C03646=1227.699,20.844,-42.507,-179.267,5.370,148.713
C03647=1227.694,21.094,-42.523,-179.265,5.371,148.713
C03648=1227.689,21.344,-42.538,-179.262,5.371,148.712
C03649=1227.684,21.593,-42.554,-179.259,5.372,148.711
C03650=1227.679,21.842,-42.569,-179.257,5.372,148.711
C03651=1227.674,22.092,-42.584,-179.255,5.372,148.710
C03652=1227.669,22.342,-42.600,-179.252,5.373,148.709
C03653=1227.664,22.591,-42.615,-179.250,5.373,148.709
C03654=1227.659,22.841,-42.630,-179.247,5.374,148.708
C03655=1227.654,23.090,-42.645,-179.244,5.374,148.707
C03656=1227.649,23.339,-42.661,-179.242,5.375,148.707
C03657=1227.644,23.589,-42.677,-179.240,5.375,148.706
C03658=1227.639,23.838,-42.692,-179.237,5.375,148.705
C03659=1227.634,24.088,-42.707,-179.234,5.376,148.705
C03660=1227.629,24.337,-42.722,-179.232,5.376,148.704
C03661=1227.625,24.587,-42.738,-179.229,5.377,148.703
C03662=1227.619,24.836,-42.754,-179.227,5.377,148.703
C03663=1227.615,25.085,-42.769,-179.224,5.377,148.702
C03664=1227.609,25.335,-42.784,-179.222,5.378,148.701
C03665=1227.604,25.585,-42.800,-179.219,5.378,148.701
C03666=1227.600,25.834,-42.815,-179.216,5.379,148.700
C03667=1227.594,26.083,-42.831,-179.214,5.379,148.699
C03668=1227.589,26.333,-42.847,-179.212,5.379,148.699
C03669=1227.585,26.583,-42.862,-179.209,5.380,148.698
C03670=1227.579,26.832,-42.878,-179.206,5.380,148.697
C03671=1227.574,27.081,-42.893,-179.204,5.381,148.697
C03672=1227.569,27.330,-42.908,-179.202,5.382,148.696
C03673=1227.565,27.581,-42.924,-179.199,5.382,148.695
C03674=1227.559,27.830,-42.940,-179.197,5.382,148.695
C03675=1227.554,28.079,-42.955,-179.194,5.382,148.694
C03676=1227.550,28.329,-42.971,-179.192,5.383,148.693
C03677=1227.544,28.579,-42.986,-179.189,5.384,148.693
C03678=1227.539,28.827,-43.002,-179.186,5.384,148.692
C03679=1227.535,29.076,-43.017,-179.184,5.385,148.691
C03680=1227.530,29.346,-43.035,-179.181,5.385,148.691
C03681=1227.524,29.615,-43.051,-179.178,5.386,148.690
C03682=1227.518,29.883,-43.068,-179.176,5.386,148.689
C03683=1227.513,30.152,-43.085,-179.173,5.387,148.688
C03684=1227.508,30.401,-43.100,-179.171,5.386,148.688
C03685=1227.503,30.651,-43.116,-179.168,5.387,148.687
C03686=1227.498,30.900,-43.132,-179.166,5.388,148.687
C03687=1227.493,31.149,-43.148,-179.163,5.388,148.686
C03688=1227.488,31.399,-43.164,-179.161,5.389,148.685
C03689=1227.483,31.648,-43.179,-179.158,5.389,148.684
C03690=1227.478,31.898,-43.195,-179.155,5.390,148.684
C03691=1227.474,32.147,-43.211,-179.153,5.390,148.683
C03692=1227.468,32.397,-43.227,-179.151,5.390,148.682
C03693=1227.463,32.647,-43.243,-179.148,5.391,148.682
C03694=1227.459,32.896,-43.258,-179.145,5.391,148.681
C03695=1227.454,33.145,-43.274,-179.143,5.392,148.680
C03696=1227.449,33.395,-43.290,-179.140,5.392,148.680
C03697=1227.444,33.644,-43.306,-179.137,5.393,148.679
C03698=1227.438,33.893,-43.321,-179.135,5.393,148.678
C03699=1227.434,34.143,-43.338,-179.133,5.393,148.678
C03700=1227.429,34.392,-43.353,-179.130,5.394,148.677
C03701=1227.424,34.642,-43.369,-179.128,5.395,148.677
C03702=1227.419,34.891,-43.385,-179.125,5.395,148.676
C03703=1227.414,35.140,-43.401,-179.123,5.396,148.675
C03704=1227.409,35.390,-43.417,-179.120,5.396,148.675
C03705=1227.404,35.640,-43.432,-179.118,5.396,148.674
C03706=1227.399,35.889,-43.449,-179.115,5.397,148.673
C03707=1227.394,36.139,-43.465,-179.113,5.397,148.673
C03708=1227.389,36.387,-43.480,-179.110,5.398,148.672
C03709=1227.385,36.637,-43.496,-179.107,5.398,148.671
C03710=1227.379,36.887,-43.512,-179.105,5.399,148.671
C03711=1227.375,37.136,-43.528,-179.102,5.399,148.670
C03712=1227.369,37.386,-43.544,-179.100,5.400,148.669
C03713=1227.364,37.635,-43.560,-179.098,5.400,148.669
C03714=1227.359,37.884,-43.576,-179.095,5.401,148.668
C03715=1227.354,38.134,-43.592,-179.092,5.401,148.667
C03716=1227.350,38.383,-43.609,-179.090,5.402,148.667
C03717=1227.344,38.633,-43.624,-179.087,5.402,148.666
C03718=1227.339,38.883,-43.640,-179.085,5.403,148.665
C03719=1227.334,39.132,-43.656,-179.082,5.403,148.665
C03720=1227.330,39.382,-43.672,-179.079,5.404,148.664
C03721=1227.324,39.631,-43.689,-179.077,5.405,148.663
C03722=1227.319,39.880,-43.704,-179.075,5.404,148.663
C03723=1227.315,40.129,-43.721,-179.072,5.405,148.662
C03724=1227.309,40.379,-43.736,-179.070,5.406,148.662
C03725=1227.305,40.628,-43.753,-179.067,5.406,148.661
C03726=1227.299,40.878,-43.769,-179.064,5.407,148.660
C03727=1227.295,41.127,-43.785,-179.062,5.407,148.659
C03728=1227.289,41.377,-43.801,-179.059,5.408,148.659
C03729=1227.285,41.626,-43.818,-179.057,5.409,148.658
C03730=1227.280,41.875,-43.833,-179.054,5.409,148.657
C03731=1227.275,42.125,-43.850,-179.052,5.409,148.657
C03732=1227.270,42.374,-43.866,-179.049,5.409,148.656
C03733=1227.265,42.624,-43.882,-179.047,5.410,148.655
C03734=1227.260,42.873,-43.898,-179.044,5.411,148.655
C03735=1227.255,43.123,-43.914,-179.042,5.411,148.654
C03736=1227.250,43.372,-43.931,-179.039,5.412,148.654
C03737=1227.246,43.622,-43.947,-179.037,5.413,148.653
C03738=1227.240,43.870,-43.963,-179.034,5.413,148.652
C03739=1227.236,44.120,-43.980,-179.031,5.414,148.652
C03740=1227.230,44.370,-43.996,-179.029,5.414,148.651
C03741=1227.225,44.619,-44.013,-179.027,5.414,148.650
C03742=1227.221,44.869,-44.028,-179.024,5.415,148.650
C03743=1227.215,45.118,-44.045,-179.022,5.416,148.649
C03744=1227.211,45.367,-44.061,-179.019,5.416,148.649
C03745=1227.206,45.617,-44.077,-179.016,5.417,148.648
C03746=1227.201,45.866,-44.094,-179.014,5.417,148.647
C03747=1227.196,46.115,-44.110,-179.011,5.418,148.646
C03748=1227.191,46.365,-44.126,-179.009,5.418,148.646
C03749=1227.185,46.614,-44.143,-179.006,5.419,148.645
C03750=1227.181,46.864,-44.160,-179.003,5.419,148.644
C03751=1227.176,47.114,-44.175,-179.001,5.420,148.644
C03752=1227.171,47.363,-44.192,-178.998,5.421,148.643
C03753=1227.167,47.612,-44.208,-178.996,5.421,148.643
C03754=1227.162,47.861,-44.225,-178.994,5.421,148.642
C03755=1227.157,48.111,-44.241,-178.991,5.422,148.641
C03756=1227.151,48.360,-44.258,-178.989,5.422,148.641
C03757=1227.146,48.610,-44.274,-178.986,5.423,148.640
C03758=1227.142,48.859,-44.291,-178.983,5.424,148.639
C03759=1227.137,49.109,-44.307,-178.981,5.424,148.639
C03760=1227.132,49.358,-44.323,-178.978,5.425,148.638
C03761=1227.127,49.608,-44.340,-178.976,5.426,148.638
C03762=1227.122,49.857,-44.357,-178.973,5.426,148.637
C03763=1227.117,50.106,-44.373,-178.971,5.427,148.636
C03764=1227.112,50.355,-44.389,-178.968,5.427,148.636
C03765=1227.107,50.605,-44.406,-178.965,5.428,148.635
C03766=1227.102,50.855,-44.423,-178.963,5.428,148.634
C03767=1227.097,51.104,-44.439,-178.961,5.428,148.634
C03768=1227.093,51.353,-44.456,-178.958,5.429,148.633
C03769=1227.088,51.603,-44.473,-178.956,5.430,148.632
C03770=1227.082,51.852,-44.490,-178.953,5.430,148.632
C03771=1227.078,52.102,-44.505,-178.951,5.431,148.631
C03772=1227.073,52.351,-44.522,-178.948,5.431,148.630
C03773=1227.067,52.600,-44.539,-178.945,5.432,148.630
C03774=1227.063,52.850,-44.556,-178.943,5.433,148.629
C03775=1227.058,53.099,-44.572,-178.940,5.433,148.628
C03776=1227.053,53.348,-44.589,-178.938,5.434,148.628
C03777=1227.048,53.598,-44.606,-178.935,5.435,148.627
C03778=1227.044,53.847,-44.623,-178.933,5.435,148.627
C03779=1227.038,54.096,-44.639,-178.930,5.436,148.626
C03780=1227.033,54.346,-44.656,-178.927,5.436,148.625
C03781=1227.029,54.595,-44.673,-178.925,5.437,148.625
C03782=1227.024,54.844,-44.689,-178.922,5.437,148.624
C03783=1227.019,55.094,-44.706,-178.920,5.438,148.624
C03784=1227.013,55.362,-44.723,-178.917,5.439,148.623
C03785=1227.008,55.631,-44.742,-178.914,5.439,148.622
C03786=1227.002,55.899,-44.760,-178.911,5.440,148.621
C03787=1226.998,56.168,-44.778,-178.909,5.440,148.621
C03788=1226.992,56.418,-44.795,-178.906,5.441,148.620
C03789=1226.987,56.666,-44.812,-178.904,5.441,148.619
C03790=1226.983,56.916,-44.828,-178.901,5.442,148.619
C03791=1226.978,57.166,-44.845,-178.899,5.443,148.618
C03792=1226.973,57.415,-44.862,-178.896,5.444,148.618
C03793=1226.967,57.664,-44.879,-178.894,5.444,148.617
C03794=1226.963,57.914,-44.896,-178.891,5.445,148.616
C03795=1226.958,58.163,-44.912,-178.888,5.445,148.616
C03796=1226.953,58.413,-44.930,-178.886,5.446,148.615
C03797=1226.948,58.662,-44.946,-178.883,5.447,148.614
C03798=1226.943,58.911,-44.964,-178.881,5.447,148.614
C03799=1226.939,59.160,-44.981,-178.878,5.448,148.613
C03800=1226.933,59.410,-44.998,-178.876,5.448,148.612
C03801=1226.928,59.659,-45.014,-178.873,5.449,148.612
C03802=1226.924,59.908,-45.031,-178.870,5.450,148.611
C03803=1226.919,60.158,-45.048,-178.868,5.451,148.611
C03804=1226.914,60.408,-45.065,-178.866,5.451,148.610
C03805=1226.909,60.656,-45.082,-178.863,5.452,148.609
C03806=1226.904,60.906,-45.099,-178.860,5.452,148.609
C03807=1226.899,61.155,-45.116,-178.858,5.453,148.608
C03808=1226.895,61.405,-45.133,-178.855,5.453,148.607
C03809=1226.889,61.655,-45.150,-178.853,5.454,148.607
C03810=1226.884,61.904,-45.167,-178.851,5.454,148.606
C03811=1226.879,62.153,-45.185,-178.848,5.455,148.606
C03812=1226.875,62.402,-45.201,-178.846,5.455,148.605
C03813=1226.870,62.652,-45.218,-178.843,5.456,148.604
C03814=1226.865,62.901,-45.235,-178.840,5.456,148.604
C03815=1226.860,63.150,-45.253,-178.838,5.457,148.603
C03816=1226.855,63.399,-45.269,-178.836,5.458,148.602
C03817=1226.850,63.649,-45.287,-178.833,5.459,148.602
C03818=1226.845,63.899,-45.303,-178.830,5.459,148.601
C03819=1226.841,64.148,-45.321,-178.828,5.460,148.600
C03820=1226.835,64.398,-45.339,-178.825,5.461,148.600
C03821=1226.830,64.646,-45.355,-178.823,5.461,148.599
C03822=1226.825,64.896,-45.373,-178.820,5.462,148.599
C03823=1226.821,65.145,-45.390,-178.818,5.462,148.598
C03824=1226.816,65.395,-45.407,-178.815,5.463,148.597
C03825=1226.811,65.644,-45.424,-178.812,5.463,148.597
C03826=1226.806,65.894,-45.441,-178.810,5.464,148.596
C03827=1226.801,66.143,-45.459,-178.808,5.465,148.596
C03828=1226.796,66.392,-45.476,-178.805,5.466,148.595
C03829=1226.791,66.641,-45.493,-178.802,5.466,148.594
C03830=1226.787,66.891,-45.510,-178.800,5.467,148.594
C03831=1226.782,67.140,-45.528,-178.798,5.468,148.593
C03832=1226.776,67.390,-45.545,-178.794,5.469,148.593
C03833=1226.772,67.639,-45.562,-178.792,5.470,148.592
C03834=1226.767,67.888,-45.580,-178.789,5.470,148.591
C03835=1226.762,68.138,-45.597,-178.786,5.471,148.591
C03836=1226.757,68.386,-45.614,-178.784,5.471,148.590
C03837=1226.752,68.636,-45.631,-178.782,5.472,148.589
C03838=1226.747,68.885,-45.649,-178.779,5.473,148.589
C03839=1226.742,69.135,-45.666,-178.776,5.474,148.588
C03840=1226.738,69.384,-45.684,-178.774,5.474,148.587
C03841=1226.732,69.634,-45.701,-178.771,5.475,148.587
C03842=1226.728,69.883,-45.718,-178.769,5.476,148.586
C03843=1226.723,70.132,-45.736,-178.766,5.476,148.586
C03844=1226.718,70.382,-45.753,-178.764,5.477,148.585
C03845=1226.714,70.631,-45.770,-178.761,5.477,148.584
C03846=1226.709,70.880,-45.788,-178.758,5.478,148.584
C03847=1226.703,71.130,-45.806,-178.756,5.479,148.583
C03848=1226.699,71.379,-45.823,-178.754,5.479,148.583
C03849=1226.694,71.629,-45.840,-178.751,5.480,148.582
C03850=1226.688,71.877,-45.858,-178.748,5.481,148.581
C03851=1226.683,72.127,-45.875,-178.746,5.481,148.581
C03852=1226.679,72.376,-45.892,-178.744,5.482,148.580
C03853=1226.674,72.626,-45.910,-178.741,5.483,148.580
C03854=1226.669,72.875,-45.928,-178.738,5.483,148.579
C03855=1226.664,73.125,-45.945,-178.736,5.484,148.578
C03856=1226.660,73.374,-45.962,-178.733,5.485,148.578
C03857=1226.655,73.623,-45.980,-178.731,5.485,148.577
C03858=1226.649,73.873,-45.998,-178.728,5.486,148.577
C03859=1226.645,74.122,-46.016,-178.726,5.487,148.576
C03860=1226.640,74.371,-46.034,-178.723,5.487,148.575
C03861=1226.635,74.620,-46.050,-178.721,5.488,148.575
C03862=1226.630,74.870,-46.068,-178.718,5.490,148.574
C03863=1226.625,75.119,-46.086,-178.715,5.490,148.573
C03864=1226.620,75.368,-46.103,-178.713,5.491,148.573
C03865=1226.615,75.618,-46.121,-178.710,5.491,148.572
C03866=1226.610,75.867,-46.139,-178.708,5.492,148.572
C03867=1226.606,76.116,-46.156,-178.705,5.493,148.571
C03868=1226.601,76.366,-46.174,-178.703,5.493,148.570
C03869=1226.596,76.615,-46.192,-178.700,5.494,148.570
C03870=1226.591,76.864,-46.209,-178.698,5.495,148.569
C03871=1226.586,77.114,-46.227,-178.695,5.496,148.569
C03872=1226.581,77.363,-46.245,-178.693,5.496,148.568
C03873=1226.577,77.612,-46.263,-178.690,5.497,148.567
C03874=1226.572,77.861,-46.280,-178.687,5.497,148.567
C03875=1226.567,78.111,-46.298,-178.685,5.498,148.566
C03876=1226.562,78.361,-46.316,-178.683,5.499,148.566
C03877=1226.557,78.610,-46.334,-178.680,5.499,148.565
C03878=1226.552,78.860,-46.351,-178.677,5.500,148.564
C03879=1226.547,79.109,-46.369,-178.675,5.502,148.564
C03880=1226.542,79.358,-46.387,-178.672,5.502,148.563
C03881=1226.537,79.607,-46.405,-178.669,5.503,148.563
C03882=1226.533,79.856,-46.423,-178.667,5.504,148.562
C03883=1226.527,80.106,-46.441,-178.665,5.505,148.561
C03884=1226.522,80.355,-46.459,-178.662,5.505,148.561
C03885=1226.518,80.604,-46.476,-178.659,5.506,148.560
C03886=1226.513,80.853,-46.494,-178.657,5.506,148.559
C03887=1226.508,81.102,-46.512,-178.655,5.507,148.559
C03888=1226.503,81.371,-46.531,-178.652,5.508,148.558
C03889=1226.497,81.640,-46.551,-178.649,5.509,148.558
C03890=1226.492,81.908,-46.570,-178.646,5.510,148.557
C03891=1226.487,82.176,-46.589,-178.643,5.510,148.556
C03892=1226.482,82.426,-46.607,-178.641,5.511,148.556
C03893=1226.477,82.675,-46.625,-178.638,5.512,148.555
C03894=1226.473,82.925,-46.644,-178.636,5.512,148.554
C03895=1226.468,83.174,-46.662,-178.633,5.514,148.554
C03896=1226.463,83.423,-46.680,-178.630,5.515,148.553
C03897=1226.458,83.672,-46.698,-178.628,5.515,148.553
C03898=1226.453,83.921,-46.716,-178.625,5.516,148.552
C03899=1226.448,84.170,-46.734,-178.623,5.517,148.552
C03900=1226.443,84.420,-46.752,-178.620,5.517,148.551
C03901=1226.439,84.670,-46.770,-178.618,5.518,148.550
C03902=1226.434,84.919,-46.788,-178.616,5.519,148.550
C03903=1226.429,85.168,-46.806,-178.613,5.519,148.549
C03904=1226.424,85.417,-46.824,-178.610,5.520,148.549
C03905=1226.419,85.666,-46.842,-178.607,5.522,148.548
C03906=1226.415,85.915,-46.860,-178.605,5.522,148.548
C03907=1226.410,86.165,-46.878,-178.602,5.523,148.547
C03908=1226.405,86.414,-46.896,-178.600,5.524,148.546
C03909=1226.400,86.664,-46.914,-178.597,5.524,148.546
C03910=1226.395,86.913,-46.933,-178.595,5.525,148.545
C03911=1226.390,87.162,-46.951,-178.592,5.526,148.545
C03912=1226.385,87.411,-46.969,-178.590,5.526,148.544
C03913=1226.381,87.661,-46.987,-178.587,5.527,148.543
C03914=1226.376,87.911,-47.005,-178.584,5.529,148.543
C03915=1226.371,88.160,-47.023,-178.582,5.529,148.542
C03916=1226.366,88.408,-47.042,-178.579,5.530,148.541
C03917=1226.361,88.657,-47.060,-178.577,5.531,148.541
C03918=1226.356,88.908,-47.079,-178.574,5.532,148.540
C03919=1226.351,89.157,-47.097,-178.572,5.532,148.540
C03920=1226.346,89.406,-47.115,-178.569,5.533,148.539
C03921=1226.342,89.655,-47.133,-178.567,5.534,148.539
C03922=1226.337,89.905,-47.151,-178.564,5.535,148.538
C03923=1226.333,90.154,-47.170,-178.561,5.536,148.537
C03924=1226.327,90.403,-47.188,-178.559,5.537,148.537
C03925=1226.322,90.652,-47.206,-178.556,5.537,148.536
C03926=1226.318,90.902,-47.225,-178.554,5.538,148.536
C03927=1226.313,91.151,-47.243,-178.551,5.538,148.535
C03928=1226.308,91.400,-47.261,-178.549,5.539,148.535
C03929=1226.303,91.649,-47.280,-178.546,5.540,148.534
C03930=1226.298,91.899,-47.298,-178.543,5.541,148.533
C03931=1226.293,92.148,-47.316,-178.541,5.542,148.533
C03932=1226.289,92.397,-47.335,-178.539,5.543,148.532
C03933=1226.283,92.646,-47.353,-178.536,5.544,148.532
C03934=1226.279,92.896,-47.372,-178.533,5.544,148.531
C03935=1226.274,93.145,-47.390,-178.531,5.545,148.531
C03936=1226.269,93.394,-47.408,-178.529,5.546,148.530
C03937=1226.264,93.644,-47.427,-178.525,5.547,148.529
C03938=1226.259,93.893,-47.445,-178.523,5.548,148.529
C03939=1226.255,94.142,-47.464,-178.521,5.549,148.528
C03940=1226.250,94.391,-47.482,-178.518,5.549,148.527
C03941=1226.245,94.641,-47.501,-178.516,5.550,148.527
C03942=1226.240,94.890,-47.520,-178.513,5.551,148.526
C03943=1226.235,95.139,-47.538,-178.510,5.552,148.526
C03944=1226.230,95.389,-47.557,-178.507,5.553,148.525
C03945=1226.226,95.638,-47.575,-178.505,5.554,148.525
C03946=1226.221,95.887,-47.593,-178.503,5.554,148.524
C03947=1226.217,96.136,-47.612,-178.500,5.555,148.523
C03948=1226.211,96.386,-47.631,-178.498,5.556,148.523
C03949=1226.206,96.634,-47.650,-178.495,5.557,148.522
C03950=1226.201,96.884,-47.669,-178.492,5.558,148.522
C03951=1226.196,97.134,-47.687,-178.490,5.559,148.521
C03952=1226.192,97.382,-47.705,-178.487,5.560,148.521
C03953=1226.187,97.632,-47.724,-178.485,5.560,148.520
C03954=1226.182,97.881,-47.743,-178.483,5.561,148.520
C03955=1226.177,98.130,-47.761,-178.480,5.562,148.519
C03956=1226.172,98.380,-47.780,-178.477,5.563,148.518
C03957=1226.168,98.629,-47.798,-178.475,5.564,148.518
C03958=1226.163,98.878,-47.818,-178.472,5.565,148.517
C03959=1226.158,99.128,-47.836,-178.470,5.565,148.517
C03960=1226.153,99.376,-47.855,-178.467,5.566,148.516
C03961=1226.148,99.626,-47.874,-178.464,5.568,148.516
C03962=1226.144,99.875,-47.892,-178.462,5.568,148.515
C03963=1226.139,100.125,-47.911,-178.459,5.569,148.514
C03964=1226.134,100.374,-47.930,-178.457,5.570,148.514
C03965=1226.129,100.623,-47.948,-178.454,5.571,148.513
C03966=1226.124,100.872,-47.968,-178.452,5.572,148.513
C03967=1226.120,101.121,-47.986,-178.449,5.573,148.512
C03968=1226.115,101.371,-48.005,-178.446,5.574,148.511
C03969=1226.110,101.620,-48.024,-178.444,5.575,148.511
C03970=1226.104,101.869,-48.043,-178.442,5.575,148.510
C03971=1226.100,102.118,-48.062,-178.439,5.576,148.510
C03972=1226.095,102.367,-48.081,-178.436,5.578,148.509
C03973=1226.091,102.617,-48.099,-178.434,5.578,148.509
C03974=1226.085,102.866,-48.119,-178.431,5.579,148.508
C03975=1226.081,103.115,-48.138,-178.429,5.580,148.508
C03976=1226.076,103.365,-48.156,-178.426,5.580,148.507
C03977=1226.071,103.613,-48.175,-178.423,5.582,148.506
C03978=1226.066,103.863,-48.195,-178.421,5.583,148.506
C03979=1226.062,104.112,-48.213,-178.418,5.583,148.505
C03980=1226.057,104.362,-48.232,-178.416,5.584,148.505
C03981=1226.052,104.610,-48.251,-178.414,5.585,148.504
C03982=1226.047,104.860,-48.270,-178.410,5.586,148.504
C03983=1226.043,105.109,-48.289,-178.408,5.587,148.503
C03984=1226.038,105.359,-48.308,-178.406,5.588,148.503
C03985=1226.033,105.607,-48.327,-178.403,5.589,148.502
C03986=1226.028,105.857,-48.346,-178.401,5.589,148.501
C03987=1226.023,106.106,-48.365,-178.398,5.591,148.501
C03988=1226.019,106.355,-48.384,-178.395,5.592,148.500
C03989=1226.013,106.604,-48.403,-178.393,5.592,148.500
C03990=1226.009,106.854,-48.422,-178.390,5.593,148.499
C03991=1226.004,107.103,-48.441,-178.387,5.595,148.499
C03992=1225.999,107.372,-48.462,-178.385,5.595,148.498
C03993=1225.993,107.640,-48.483,-178.383,5.596,148.497
C03994=1225.989,107.909,-48.503,-178.379,5.598,148.497
C03995=1225.983,108.176,-48.523,-178.377,5.598,148.496
C03996=1225.979,108.426,-48.543,-178.374,5.599,148.496
C03997=1225.973,108.675,-48.562,-178.371,5.601,148.495
C03998=1225.969,108.925,-48.581,-178.369,5.601,148.495
C03999=1225.964,109.174,-48.600,-178.367,5.602,148.494
C04000=1225.959,109.423,-48.620,-178.364,5.603,148.493
C04001=1225.954,109.672,-48.638,-178.361,5.604,148.493
C04002=1225.950,109.921,-48.658,-178.359,5.605,148.492
C04003=1225.945,110.171,-48.678,-178.356,5.606,148.492
C04004=1225.940,110.419,-48.696,-178.354,5.606,148.491
C04005=1225.935,110.669,-48.716,-178.351,5.607,148.491
C04006=1225.930,110.918,-48.735,-178.348,5.609,148.490
C04007=1225.926,111.167,-48.754,-178.346,5.610,148.490
C04008=1225.921,111.416,-48.774,-178.344,5.610,148.489
C04009=1225.916,111.666,-48.793,-178.341,5.611,148.488
C04010=1225.912,111.915,-48.812,-178.338,5.613,148.488
C04011=1225.907,112.164,-48.832,-178.336,5.613,148.487
C04012=1225.902,112.413,-48.851,-178.333,5.614,148.487
C04013=1225.897,112.662,-48.871,-178.331,5.615,148.486
C04014=1225.893,112.911,-48.890,-178.328,5.616,148.486
C04015=1225.888,113.161,-48.909,-178.326,5.617,148.485
C04016=1225.882,113.410,-48.929,-178.323,5.618,148.485
C04017=1225.878,113.659,-48.948,-178.321,5.619,148.484
C04018=1225.873,113.908,-48.967,-178.318,5.620,148.484
C04019=1225.868,114.158,-48.987,-178.315,5.621,148.483
C04020=1225.864,114.407,-49.006,-178.313,5.622,148.483
C04021=1225.858,114.656,-49.026,-178.310,5.623,148.482
C04022=1225.854,114.906,-49.045,-178.308,5.624,148.481
C04023=1225.849,115.154,-49.064,-178.305,5.625,148.481
C04024=1225.844,115.404,-49.084,-178.302,5.626,148.480
C04025=1225.839,115.653,-49.103,-178.300,5.627,148.480
C04026=1225.834,115.902,-49.123,-178.297,5.628,148.479
C04027=1225.829,116.152,-49.142,-178.295,5.629,148.479
C04028=1225.825,116.401,-49.163,-178.292,5.630,148.478
C04029=1225.820,116.649,-49.181,-178.289,5.631,148.477
C04030=1225.816,116.899,-49.201,-178.287,5.632,148.477
C04031=1225.811,117.148,-49.221,-178.284,5.633,148.476
C04032=1225.805,117.397,-49.240,-178.282,5.634,148.476
C04033=1225.801,117.647,-49.260,-178.279,5.635,148.475
C04034=1225.796,117.896,-49.280,-178.277,5.636,148.475
C04035=1225.791,118.145,-49.299,-178.274,5.637,148.474
C04036=1225.786,118.394,-49.319,-178.271,5.638,148.474
C04037=1225.782,118.643,-49.338,-178.269,5.639,148.473
C04038=1225.777,118.892,-49.357,-178.267,5.640,148.473
C04039=1225.772,119.141,-49.378,-178.264,5.641,148.472
C04040=1225.768,119.391,-49.397,-178.261,5.642,148.472
C04041=1225.763,119.640,-49.417,-178.259,5.643,148.471
C04042=1225.758,119.889,-49.436,-178.257,5.644,148.471
C04043=1225.753,120.138,-49.457,-178.253,5.645,148.470
C04044=1225.748,120.388,-49.476,-178.251,5.646,148.470
C04045=1225.743,120.637,-49.495,-178.249,5.647,148.469
C04046=1225.739,120.886,-49.516,-178.246,5.649,148.469
C04047=1225.734,121.135,-49.536,-178.243,5.649,148.468
C04048=1225.729,121.385,-49.555,-178.241,5.650,148.467
C04049=1225.724,121.633,-49.575,-178.239,5.651,148.467
C04050=1225.719,121.883,-49.595,-178.235,5.652,148.466
C04051=1225.715,122.132,-49.614,-178.233,5.653,148.466
C04052=1225.710,122.381,-49.635,-178.231,5.654,148.465
C04053=1225.705,122.630,-49.654,-178.228,5.656,148.465
C04054=1225.700,122.879,-49.674,-178.225,5.656,148.464
C04055=1225.696,123.128,-49.694,-178.223,5.657,148.464
C04056=1225.691,123.378,-49.714,-178.220,5.659,148.463
C04057=1225.686,123.626,-49.734,-178.218,5.660,148.463
C04058=1225.681,123.876,-49.753,-178.215,5.660,148.462
C04059=1225.676,124.125,-49.773,-178.212,5.662,148.461
C04060=1225.672,124.374,-49.794,-178.210,5.663,148.461
C04061=1225.667,124.624,-49.813,-178.208,5.663,148.460
C04062=1225.662,124.872,-49.833,-178.205,5.664,148.460
C04063=1225.657,125.122,-49.853,-178.202,5.666,148.459
C04064=1225.653,125.371,-49.873,-178.200,5.667,148.459
C04065=1225.648,125.620,-49.893,-178.198,5.667,148.458
C04066=1225.644,125.869,-49.913,-178.195,5.669,148.458
C04067=1225.638,126.118,-49.933,-178.192,5.670,148.457
C04068=1225.634,126.367,-49.953,-178.190,5.671,148.457
C04069=1225.629,126.617,-49.973,-178.187,5.672,148.456
C04070=1225.625,126.865,-49.993,-178.185,5.673,148.456
C04071=1225.620,127.115,-50.013,-178.182,5.674,148.455
C04072=1225.615,127.364,-50.034,-178.179,5.675,148.455
C04073=1225.610,127.613,-50.053,-178.177,5.676,148.454
C04074=1225.605,127.862,-50.073,-178.174,5.677,148.454
C04075=1225.600,128.112,-50.093,-178.172,5.679,148.453
C04076=1225.596,128.361,-50.113,-178.169,5.679,148.453
C04077=1225.592,128.610,-50.134,-178.167,5.680,148.452
C04078=1225.587,128.859,-50.153,-178.164,5.682,148.452
C04079=1225.581,129.108,-50.174,-178.162,5.683,148.451
C04080=1225.576,129.357,-50.194,-178.159,5.684,148.451
C04081=1225.572,129.606,-50.214,-178.156,5.685,148.450
C04082=1225.567,129.855,-50.234,-178.154,5.686,148.449
C04083=1225.563,130.105,-50.254,-178.151,5.688,148.449
C04084=1225.558,130.354,-50.274,-178.149,5.688,148.448
C04085=1225.553,130.603,-50.295,-178.146,5.689,148.448
C04086=1225.548,130.853,-50.315,-178.143,5.691,148.447
C04087=1225.544,131.101,-50.335,-178.141,5.692,148.447
C04088=1225.539,131.350,-50.355,-178.139,5.692,148.446
C04089=1225.534,131.599,-50.375,-178.136,5.694,148.446
C04090=1225.529,131.849,-50.396,-178.133,5.695,148.445
C04091=1225.524,132.098,-50.416,-178.131,5.696,148.445
C04092=1225.520,132.346,-50.437,-178.128,5.697,148.444
C04093=1225.515,132.596,-50.456,-178.126,5.698,148.444
C04094=1225.510,132.845,-50.477,-178.123,5.700,148.443
C04095=1225.506,133.094,-50.498,-178.121,5.701,148.443
C04096=1225.500,133.363,-50.519,-178.118,5.701,148.442
C04097=1225.495,133.631,-50.541,-178.115,5.703,148.442
C04098=1225.490,133.900,-50.563,-178.112,5.705,148.441
C04099=1225.485,134.169,-50.586,-178.110,5.705,148.441
C04100=1225.481,134.418,-50.606,-178.106,5.707,148.440
C04101=1225.476,134.667,-50.626,-178.104,5.708,148.440
C04102=1225.471,134.916,-50.647,-178.102,5.708,148.439
C04103=1225.466,135.165,-50.667,-178.099,5.710,148.439
C04104=1225.461,135.414,-50.687,-178.096,5.711,148.438
C04105=1225.456,135.663,-50.708,-178.094,5.712,148.438
C04106=1225.452,135.912,-50.728,-178.092,5.713,148.437
C04107=1225.447,136.161,-50.749,-178.089,5.714,148.437
C04108=1225.442,136.411,-50.770,-178.086,5.716,148.436
C04109=1225.438,136.660,-50.790,-178.084,5.717,148.436
C04110=1225.433,136.909,-50.810,-178.082,5.717,148.435
C04111=1225.428,137.158,-50.831,-178.078,5.719,148.435
C04112=1225.423,137.407,-50.851,-178.076,5.720,148.434
C04113=1225.419,137.656,-50.871,-178.073,5.721,148.434
C04114=1225.414,137.906,-50.892,-178.071,5.722,148.433
C04115=1225.409,138.155,-50.913,-178.068,5.723,148.433
C04116=1225.404,138.404,-50.934,-178.066,5.725,148.432
C04117=1225.400,138.653,-50.954,-178.063,5.725,148.432
C04118=1225.394,138.902,-50.975,-178.061,5.727,148.431
C04119=1225.390,139.151,-50.995,-178.058,5.728,148.431
C04120=1225.385,139.400,-51.016,-178.056,5.729,148.430
C04121=1225.380,139.649,-51.037,-178.053,5.730,148.430
C04122=1225.376,139.899,-51.057,-178.051,5.731,148.429
C04123=1225.371,140.148,-51.078,-178.048,5.733,148.429
C04124=1225.367,140.397,-51.099,-178.045,5.734,148.428
C04125=1225.362,140.646,-51.120,-178.043,5.735,148.428
C04126=1225.357,140.895,-51.140,-178.040,5.736,148.427
C04127=1225.352,141.144,-51.161,-178.038,5.737,148.427
C04128=1225.348,141.393,-51.181,-178.035,5.739,148.426
C04129=1225.343,141.642,-51.203,-178.033,5.740,148.426
C04130=1225.338,141.891,-51.224,-178.030,5.740,148.425
C04131=1225.334,142.140,-51.244,-178.027,5.742,148.425
C04132=1225.329,142.389,-51.265,-178.025,5.743,148.424
C04133=1225.324,142.638,-51.285,-178.022,5.745,148.424
C04134=1225.319,142.887,-51.306,-178.020,5.746,148.423
C04135=1225.314,143.137,-51.327,-178.017,5.747,148.423
C04136=1225.310,143.386,-51.348,-178.015,5.748,148.422
C04137=1225.305,143.635,-51.370,-178.012,5.749,148.422
C04138=1225.301,143.884,-51.390,-178.009,5.750,148.421
C04139=1225.296,144.133,-51.411,-178.007,5.751,148.421
C04140=1225.291,144.382,-51.431,-178.004,5.753,148.420
C04141=1225.286,144.631,-51.452,-178.002,5.754,148.420
C04142=1225.282,144.880,-51.473,-177.999,5.755,148.419
C04143=1225.277,145.129,-51.494,-177.997,5.756,148.419
C04144=1225.272,145.378,-51.515,-177.994,5.758,148.418
C04145=1225.268,145.628,-51.536,-177.992,5.759,148.418
C04146=1225.263,145.877,-51.558,-177.989,5.759,148.417
C04147=1225.258,146.125,-51.578,-177.986,5.761,148.417
C04148=1225.253,146.375,-51.599,-177.984,5.762,148.416
C04149=1225.248,146.624,-51.620,-177.981,5.764,148.416
C04150=1225.244,146.872,-51.641,-177.979,5.765,148.415
C04151=1225.239,147.122,-51.662,-177.976,5.766,148.415
C04152=1225.235,147.371,-51.683,-177.974,5.767,148.414
C04153=1225.230,147.620,-51.705,-177.971,5.769,148.414
C04154=1225.225,147.869,-51.725,-177.968,5.770,148.413
C04155=1225.220,148.118,-51.746,-177.966,5.771,148.413
C04156=1225.216,148.367,-51.768,-177.963,5.772,148.412
C04157=1225.211,148.617,-51.789,-177.961,5.773,148.412
C04158=1225.207,148.866,-51.809,-177.958,5.775,148.411
C04159=1225.202,149.114,-51.831,-177.956,5.776,148.411
C04160=1225.196,149.364,-51.852,-177.953,5.777,148.411
C04161=1225.192,149.612,-51.872,-177.951,5.778,148.410
C04162=1225.188,149.862,-51.894,-177.948,5.780,148.410
C04163=1225.183,150.111,-51.915,-177.945,5.780,148.409
C04164=1225.178,150.360,-51.937,-177.943,5.782,148.409
C04165=1225.173,150.609,-51.957,-177.940,5.783,148.408
C04166=1225.168,150.857,-51.979,-177.937,5.785,148.408
C04167=1225.164,151.107,-52.000,-177.935,5.786,148.407
C04168=1225.159,151.356,-52.022,-177.932,5.787,148.407
C04169=1225.155,151.605,-52.042,-177.930,5.788,148.406
C04170=1225.150,151.853,-52.064,-177.927,5.790,148.406
C04171=1225.145,152.103,-52.085,-177.925,5.791,148.405
C04172=1225.140,152.352,-52.107,-177.922,5.793,148.405
C04173=1225.136,152.601,-52.127,-177.920,5.793,148.405
C04174=1225.131,152.850,-52.149,-177.917,5.795,148.404
C04175=1225.126,153.100,-52.170,-177.915,5.796,148.404
C04176=1225.121,153.348,-52.192,-177.912,5.797,148.403
C04177=1225.116,153.598,-52.213,-177.909,5.798,148.403
C04178=1225.112,153.846,-52.234,-177.907,5.799,148.402
C04179=1225.108,154.096,-52.256,-177.904,5.801,148.402
C04180=1225.103,154.344,-52.277,-177.902,5.802,148.401
C04181=1225.098,154.594,-52.298,-177.899,5.803,148.401
C04182=1225.093,154.842,-52.320,-177.897,5.804,148.400
C04183=1225.088,155.092,-52.342,-177.894,5.806,148.400
C04184=1225.084,155.341,-52.362,-177.892,5.807,148.399
C04185=1225.079,155.589,-52.384,-177.889,5.809,148.399
C04186=1225.075,155.839,-52.406,-177.887,5.810,148.398
C04187=1225.070,156.088,-52.427,-177.884,5.811,148.398
C04188=1225.065,156.337,-52.449,-177.881,5.813,148.397
C04189=1225.061,156.586,-52.471,-177.879,5.814,148.397
C04190=1225.055,156.835,-52.492,-177.876,5.815,148.396
C04191=1225.050,157.084,-52.513,-177.874,5.816,148.396
C04192=1225.047,157.333,-52.535,-177.870,5.818,148.396
C04193=1225.042,157.582,-52.556,-177.868,5.819,148.395
C04194=1225.037,157.831,-52.577,-177.866,5.821,148.395
C04195=1225.033,158.080,-52.600,-177.863,5.821,148.394
C04196=1225.028,158.329,-52.621,-177.860,5.823,148.394
C04197=1225.023,158.578,-52.642,-177.858,5.824,148.393
C04198=1225.018,158.827,-52.664,-177.855,5.826,148.393
C04199=1225.013,159.076,-52.686,-177.853,5.827,148.392
C04200=1225.008,159.345,-52.709,-177.850,5.828,148.392
C04201=1225.003,159.614,-52.732,-177.847,5.830,148.391
C04202=1224.998,159.883,-52.756,-177.845,5.831,148.391
C04203=1224.993,160.152,-52.779,-177.842,5.832,148.390
C04204=1224.989,160.401,-52.801,-177.839,5.834,148.390
C04205=1224.984,160.650,-52.823,-177.837,5.835,148.389
C04206=1224.979,160.899,-52.844,-177.834,5.837,148.389
C04207=1224.975,161.148,-52.866,-177.832,5.838,148.389
C04208=1224.970,161.397,-52.887,-177.829,5.839,148.388
C04209=1224.966,161.647,-52.909,-177.827,5.840,148.388
C04210=1224.961,161.895,-52.931,-177.824,5.842,148.387
C04211=1224.956,162.144,-52.953,-177.822,5.843,148.387
C04212=1224.952,162.393,-52.975,-177.819,5.845,148.386
C04213=1224.946,162.642,-52.997,-177.816,5.846,148.386
C04214=1224.942,162.892,-53.019,-177.814,5.847,148.385
C04215=1224.937,163.140,-53.041,-177.811,5.849,148.385
C04216=1224.933,163.390,-53.063,-177.809,5.850,148.385
C04217=1224.928,163.638,-53.084,-177.806,5.851,148.384
C04218=1224.923,163.887,-53.106,-177.804,5.852,148.384
C04219=1224.919,164.136,-53.128,-177.801,5.854,148.383
C04220=1224.914,164.385,-53.150,-177.798,5.855,148.383
C04221=1224.909,164.634,-53.172,-177.796,5.857,148.382
C04222=1224.905,164.883,-53.194,-177.793,5.858,148.382
C04223=1224.900,165.132,-53.216,-177.790,5.859,148.381
C04224=1224.895,165.381,-53.237,-177.788,5.861,148.381
C04225=1224.890,165.630,-53.260,-177.786,5.862,148.381
C04226=1224.886,165.879,-53.282,-177.783,5.863,148.380
C04227=1224.881,166.128,-53.304,-177.780,5.864,148.380
C04228=1224.876,166.377,-53.325,-177.778,5.866,148.379
C04229=1224.872,166.626,-53.347,-177.775,5.868,148.379
C04230=1224.867,166.875,-53.369,-177.773,5.869,148.378
C04231=1224.863,167.124,-53.391,-177.770,5.871,148.378
C04232=1224.857,167.373,-53.413,-177.768,5.872,148.377
C04233=1224.853,167.623,-53.436,-177.765,5.873,148.377
C04234=1224.848,167.871,-53.457,-177.763,5.874,148.376
C04235=1224.844,168.121,-53.479,-177.760,5.876,148.376
C04236=1224.839,168.369,-53.502,-177.757,5.877,148.376
C04237=1224.834,168.618,-53.524,-177.755,5.878,148.375
C04238=1224.830,168.867,-53.546,-177.752,5.880,148.375
C04239=1224.825,169.116,-53.568,-177.750,5.881,148.374
C04240=1224.820,169.365,-53.590,-177.747,5.883,148.374
C04241=1224.815,169.615,-53.612,-177.744,5.884,148.373
C04242=1224.811,169.863,-53.635,-177.742,5.885,148.373
C04243=1224.807,170.112,-53.657,-177.739,5.887,148.372
C04244=1224.802,170.361,-53.678,-177.737,5.888,148.372
C04245=1224.797,170.610,-53.701,-177.734,5.890,148.372
C04246=1224.793,170.859,-53.724,-177.731,5.892,148.371
C04247=1224.788,171.108,-53.746,-177.729,5.892,148.371
C04248=1224.784,171.357,-53.768,-177.726,5.894,148.370
C04249=1224.778,171.606,-53.790,-177.724,5.895,148.370
C04250=1224.774,171.855,-53.813,-177.721,5.897,148.370
C04251=1224.769,172.103,-53.834,-177.718,5.898,148.369
C04252=1224.764,172.353,-53.857,-177.716,5.899,148.369
C04253=1224.760,172.602,-53.879,-177.714,5.901,148.368
C04254=1224.755,172.850,-53.901,-177.711,5.902,148.368
C04255=1224.750,173.100,-53.924,-177.708,5.904,148.367
C04256=1224.745,173.349,-53.946,-177.706,5.906,148.367
C04257=1224.741,173.597,-53.969,-177.704,5.907,148.367
C04258=1224.736,173.847,-53.991,-177.700,5.908,148.366
C04259=1224.732,174.095,-54.014,-177.698,5.910,148.366
C04260=1224.728,174.344,-54.036,-177.696,5.911,148.365
C04261=1224.722,174.593,-54.058,-177.693,5.913,148.365
C04262=1224.718,174.842,-54.081,-177.690,5.913,148.364
C04263=1224.714,175.091,-54.103,-177.688,5.915,148.364
C04264=1224.709,175.340,-54.126,-177.685,5.917,148.364
C04265=1224.704,175.589,-54.148,-177.683,5.918,148.363
C04266=1224.699,175.839,-54.170,-177.680,5.920,148.363
C04267=1224.695,176.087,-54.193,-177.677,5.921,148.362
C04268=1224.690,176.336,-54.215,-177.675,5.922,148.362
C04269=1224.686,176.585,-54.238,-177.673,5.924,148.362
C04270=1224.681,176.834,-54.260,-177.670,5.925,148.361
C04271=1224.676,177.083,-54.283,-177.667,5.927,148.361
C04272=1224.672,177.332,-54.305,-177.665,5.929,148.360
C04273=1224.667,177.580,-54.328,-177.663,5.930,148.360
C04274=1224.662,177.830,-54.350,-177.660,5.931,148.359
C04275=1224.658,178.079,-54.374,-177.657,5.933,148.359
C04276=1224.653,178.327,-54.395,-177.655,5.934,148.359
C04277=1224.648,178.576,-54.419,-177.652,5.936,148.358
C04278=1224.644,178.825,-54.441,-177.649,5.938,148.358
C04279=1224.638,179.074,-54.464,-177.647,5.938,148.357
C04280=1224.635,179.323,-54.487,-177.644,5.940,148.357
C04281=1224.629,179.573,-54.509,-177.642,5.942,148.356
C04282=1224.626,179.821,-54.532,-177.639,5.943,148.356
C04283=1224.620,180.070,-54.554,-177.637,5.945,148.356
C04284=1224.616,180.319,-54.577,-177.634,5.946,148.355
C04285=1224.611,180.568,-54.600,-177.632,5.947,148.355
C04286=1224.606,180.817,-54.622,-177.629,5.949,148.354
C04287=1224.602,181.066,-54.645,-177.626,5.951,148.354
C04288=1224.598,181.314,-54.668,-177.624,5.952,148.353
C04289=1224.593,181.564,-54.691,-177.621,5.953,148.353
C04290=1224.588,181.812,-54.713,-177.618,5.955,148.353
C04291=1224.583,182.061,-54.737,-177.616,5.956,148.352
C04292=1224.578,182.311,-54.759,-177.614,5.958,148.352
C04293=1224.574,182.559,-54.782,-177.610,5.960,148.351
C04294=1224.569,182.808,-54.805,-177.608,5.961,148.351
C04295=1224.565,183.056,-54.828,-177.606,5.962,148.351
C04296=1224.560,183.306,-54.850,-177.603,5.964,148.350
C04297=1224.556,183.555,-54.874,-177.601,5.965,148.350
C04298=1224.552,183.804,-54.896,-177.598,5.967,148.349
C04299=1224.546,184.052,-54.919,-177.595,5.969,148.349
C04300=1224.542,184.301,-54.942,-177.593,5.970,148.349
C04301=1224.537,184.551,-54.965,-177.590,5.972,148.348
C04302=1224.533,184.800,-54.988,-177.588,5.973,148.348
C04303=1224.529,185.048,-55.011,-177.585,5.974,148.347
C04304=1224.523,185.318,-55.036,-177.583,5.976,148.347
C04305=1224.518,185.588,-55.061,-177.580,5.978,148.347
C04306=1224.513,185.857,-55.086,-177.577,5.979,148.346
C04307=1224.508,186.127,-55.111,-177.574,5.981,148.346
C04308=1224.503,186.376,-55.134,-177.572,5.983,148.345
C04309=1224.499,186.624,-55.156,-177.569,5.984,148.345
C04310=1224.494,186.873,-55.180,-177.566,5.985,148.344
C04311=1224.489,187.122,-55.203,-177.564,5.987,148.344
C04312=1224.485,187.371,-55.226,-177.561,5.989,148.344
C04313=1224.481,187.620,-55.249,-177.559,5.990,148.343
C04314=1224.476,187.869,-55.273,-177.556,5.992,148.343
C04315=1224.471,188.117,-55.295,-177.554,5.994,148.343
C04316=1224.467,188.366,-55.318,-177.551,5.994,148.342
C04317=1224.462,188.616,-55.341,-177.548,5.996,148.342
C04318=1224.457,188.865,-55.364,-177.546,5.998,148.341
C04319=1224.452,189.114,-55.388,-177.543,6.000,148.341
C04320=1224.448,189.363,-55.411,-177.541,6.001,148.341
C04321=1224.444,189.612,-55.434,-177.538,6.003,148.340
C04322=1224.439,189.861,-55.457,-177.535,6.004,148.340
C04323=1224.434,190.108,-55.481,-177.533,6.005,148.339
C04324=1224.429,190.357,-55.504,-177.531,6.007,148.339
C04325=1224.425,190.606,-55.528,-177.528,6.009,148.339
C04326=1224.421,190.855,-55.550,-177.525,6.011,148.338
C04327=1224.416,191.104,-55.574,-177.523,6.012,148.338
C04328=1224.411,191.353,-55.597,-177.520,6.013,148.337
C04329=1224.407,191.602,-55.620,-177.517,6.015,148.337
C04330=1224.402,191.851,-55.644,-177.515,6.017,148.337
C04331=1224.397,192.100,-55.667,-177.513,6.018,148.336
C04332=1224.392,192.349,-55.690,-177.510,6.020,148.336
C04333=1224.389,192.598,-55.713,-177.507,6.022,148.336
C04334=1224.384,192.847,-55.737,-177.505,6.024,148.335
C04335=1224.379,193.095,-55.761,-177.502,6.024,148.335
C04336=1224.374,193.344,-55.784,-177.499,6.026,148.334
C04337=1224.369,193.593,-55.807,-177.497,6.028,148.334
C04338=1224.365,193.842,-55.830,-177.494,6.030,148.334
C04339=1224.360,194.091,-55.854,-177.492,6.031,148.333
C04340=1224.356,194.339,-55.878,-177.489,6.033,148.333
C04341=1224.351,194.588,-55.901,-177.487,6.035,148.333
C04342=1224.346,194.837,-55.925,-177.484,6.036,148.332
C04343=1224.342,195.086,-55.948,-177.482,6.037,148.332
C04344=1224.338,195.335,-55.971,-177.479,6.039,148.331
C04345=1224.333,195.583,-55.995,-177.476,6.041,148.331
C04346=1224.328,195.833,-56.018,-177.474,6.043,148.331
C04347=1224.324,196.082,-56.041,-177.472,6.044,148.330
C04348=1224.319,196.330,-56.065,-177.469,6.045,148.330
C04349=1224.315,196.579,-56.089,-177.466,6.047,148.329
C04350=1224.310,196.828,-56.112,-177.464,6.049,148.329
C04351=1224.306,197.076,-56.136,-177.461,6.050,148.329
C04352=1224.301,197.325,-56.160,-177.458,6.052,148.328
C04353=1224.296,197.574,-56.183,-177.456,6.054,148.328
C04354=1224.292,197.823,-56.207,-177.453,6.055,148.328
C04355=1224.287,198.072,-56.230,-177.451,6.057,148.327
C04356=1224.282,198.321,-56.254,-177.448,6.058,148.327
C04357=1224.278,198.569,-56.278,-177.446,6.060,148.326
C04358=1224.273,198.818,-56.301,-177.443,6.062,148.326
C04359=1224.268,199.068,-56.325,-177.441,6.064,148.326
C04360=1224.264,199.317,-56.350,-177.438,6.064,148.325
C04361=1224.259,199.566,-56.373,-177.435,6.066,148.325
C04362=1224.255,199.814,-56.397,-177.433,6.068,148.324
C04363=1224.250,200.063,-56.420,-177.430,6.070,148.324
C04364=1224.246,200.312,-56.444,-177.427,6.072,148.324
C04365=1224.241,200.561,-56.468,-177.425,6.073,148.323
C04366=1224.237,200.809,-56.492,-177.423,6.075,148.323
C04367=1224.232,201.058,-56.515,-177.420,6.077,148.323
C04368=1224.228,201.307,-56.539,-177.417,6.078,148.322
C04369=1224.223,201.556,-56.563,-177.415,6.080,148.322
C04370=1224.218,201.804,-56.587,-177.413,6.081,148.322
C04371=1224.213,202.053,-56.611,-177.410,6.083,148.321
C04372=1224.209,202.303,-56.635,-177.407,6.085,148.321
C04373=1224.205,202.552,-56.659,-177.404,6.086,148.320
C04374=1224.200,202.800,-56.683,-177.402,6.088,148.320
C04375=1224.196,203.049,-56.706,-177.400,6.089,148.320
C04376=1224.191,203.297,-56.730,-177.397,6.091,148.319
C04377=1224.186,203.546,-56.755,-177.394,6.093,148.319
C04378=1224.181,203.795,-56.778,-177.392,6.095,148.319
C04379=1224.177,204.044,-56.802,-177.389,6.097,148.318
C04380=1224.173,204.293,-56.826,-177.387,6.098,148.318
C04381=1224.168,204.542,-56.850,-177.384,6.100,148.318
C04382=1224.163,204.790,-56.875,-177.382,6.101,148.317
C04383=1224.159,205.040,-56.898,-177.379,6.103,148.317
C04384=1224.154,205.288,-56.922,-177.376,6.105,148.317
C04385=1224.150,205.536,-56.946,-177.373,6.107,148.316
C04386=1224.145,205.786,-56.970,-177.371,6.108,148.316
C04387=1224.141,206.035,-56.995,-177.369,6.110,148.315
C04388=1224.136,206.283,-57.019,-177.366,6.111,148.315
C04389=1224.132,206.532,-57.043,-177.363,6.113,148.315
C04390=1224.126,206.781,-57.067,-177.361,6.115,148.314
C04391=1224.122,207.029,-57.091,-177.358,6.117,148.314
C04392=1224.118,207.278,-57.115,-177.356,6.118,148.314
C04393=1224.114,207.527,-57.139,-177.353,6.120,148.313
C04394=1224.108,207.776,-57.163,-177.351,6.122,148.313
C04395=1224.104,208.025,-57.187,-177.348,6.124,148.313
C04396=1224.100,208.273,-57.211,-177.345,6.125,148.312
C04397=1224.095,208.523,-57.236,-177.343,6.127,148.312
C04398=1224.090,208.772,-57.260,-177.341,6.128,148.312
C04399=1224.086,209.020,-57.284,-177.338,6.130,148.311
C04400=1224.081,209.269,-57.308,-177.335,6.132,148.311
C04401=1224.077,209.518,-57.333,-177.333,6.134,148.311
C04402=1224.073,209.766,-57.357,-177.330,6.136,148.310
C04403=1224.068,210.015,-57.382,-177.328,6.138,148.310
C04404=1224.063,210.263,-57.406,-177.325,6.139,148.310
C04405=1224.058,210.513,-57.430,-177.323,6.140,148.309
C04406=1224.054,210.762,-57.454,-177.320,6.142,148.309
C04407=1224.049,211.010,-57.478,-177.318,6.144,148.309
C04408=1224.044,211.280,-57.505,-177.314,6.146,148.308
C04409=1224.039,211.551,-57.532,-177.312,6.147,148.308
C04410=1224.035,211.821,-57.559,-177.309,6.150,148.307
C04411=1224.029,212.092,-57.585,-177.306,6.152,148.307
C04412=1224.025,212.341,-57.609,-177.303,6.154,148.307
C04413=1224.020,212.589,-57.633,-177.301,6.155,148.306
C04414=1224.016,212.838,-57.658,-177.299,6.157,148.306
C04415=1224.011,213.087,-57.682,-177.296,6.159,148.306
C04416=1224.006,213.336,-57.707,-177.293,6.160,148.305
C04417=1224.003,213.585,-57.731,-177.291,6.162,148.305
C04418=1223.997,213.833,-57.756,-177.288,6.164,148.305
C04419=1223.993,214.082,-57.780,-177.285,6.166,148.304
C04420=1223.988,214.331,-57.805,-177.283,6.168,148.304
C04421=1223.984,214.579,-57.830,-177.281,6.169,148.304
C04422=1223.979,214.828,-57.854,-177.278,6.171,148.303
C04423=1223.975,215.077,-57.879,-177.275,6.173,148.303
C04424=1223.970,215.326,-57.903,-177.273,6.174,148.303
C04425=1223.966,215.574,-57.927,-177.270,6.176,148.302
C04426=1223.961,215.823,-57.953,-177.268,6.178,148.302
C04427=1223.957,216.072,-57.977,-177.265,6.180,148.302
C04428=1223.952,216.321,-58.001,-177.262,6.182,148.301
C04429=1223.947,216.570,-58.026,-177.260,6.184,148.301
C04430=1223.943,216.818,-58.051,-177.257,6.186,148.301
C04431=1223.938,217.067,-58.076,-177.255,6.187,148.300
C04432=1223.934,217.316,-58.100,-177.252,6.189,148.300
C04433=1223.929,217.564,-58.125,-177.250,6.190,148.300
C04434=1223.925,217.813,-58.149,-177.247,6.192,148.299
C04435=1223.921,218.062,-58.175,-177.244,6.194,148.299
C04436=1223.915,218.310,-58.199,-177.242,6.196,148.299
C04437=1223.912,218.559,-58.224,-177.239,6.198,148.298
C04438=1223.907,218.808,-58.248,-177.237,6.200,148.298
C04439=1223.903,219.057,-58.274,-177.234,6.202,148.298
C04440=1223.898,219.305,-58.298,-177.231,6.203,148.297
C04441=1223.893,219.554,-58.323,-177.229,6.204,148.297
C04442=1223.889,219.803,-58.347,-177.227,6.206,148.297
C04443=1223.884,220.051,-58.373,-177.224,6.208,148.296
C04444=1223.880,220.301,-58.398,-177.221,6.210,148.296
C04445=1223.875,220.549,-58.422,-177.219,6.212,148.296
C04446=1223.870,220.797,-58.447,-177.216,6.214,148.295
C04447=1223.866,221.047,-58.472,-177.213,6.216,148.295
C04448=1223.861,221.295,-58.496,-177.211,6.217,148.295
C04449=1223.857,221.544,-58.522,-177.208,6.219,148.294
C04450=1223.852,221.793,-58.547,-177.206,6.221,148.294
C04451=1223.849,222.041,-58.572,-177.203,6.223,148.294
C04452=1223.844,222.290,-58.597,-177.200,6.225,148.293
C04453=1223.839,222.539,-58.622,-177.198,6.226,148.293
C04454=1223.834,222.787,-58.647,-177.196,6.228,148.293
C04455=1223.830,223.036,-58.671,-177.193,6.230,148.293
C04456=1223.826,223.285,-58.697,-177.191,6.232,148.292
C04457=1223.821,223.534,-58.722,-177.188,6.234,148.292
C04458=1223.816,223.782,-58.747,-177.186,6.236,148.292
C04459=1223.812,224.031,-58.772,-177.183,6.237,148.291
C04460=1223.808,224.279,-58.797,-177.180,6.239,148.291
C04461=1223.803,224.529,-58.822,-177.178,6.241,148.291
C04462=1223.798,224.777,-58.848,-177.175,6.243,148.290
C04463=1223.794,225.026,-58.873,-177.172,6.245,148.290
C04464=1223.790,225.274,-58.897,-177.170,6.247,148.290
C04465=1223.785,225.523,-58.922,-177.167,6.249,148.289
C04466=1223.780,225.772,-58.948,-177.165,6.250,148.289
C04467=1223.776,226.021,-58.973,-177.163,6.251,148.289
C04468=1223.771,226.269,-58.998,-177.160,6.253,148.288
C04469=1223.766,226.519,-59.023,-177.158,6.256,148.288
C04470=1223.762,226.766,-59.048,-177.155,6.257,148.288
C04471=1223.758,227.015,-59.074,-177.153,6.259,148.288
C04472=1223.753,227.264,-59.098,-177.150,6.261,148.287
C04473=1223.749,227.513,-59.124,-177.147,6.263,148.287
C04474=1223.744,227.761,-59.150,-177.145,6.265,148.287
C04475=1223.739,228.010,-59.175,-177.142,6.267,148.286
C04476=1223.735,228.259,-59.200,-177.139,6.269,148.286
C04477=1223.730,228.507,-59.226,-177.137,6.270,148.286
C04478=1223.726,228.756,-59.250,-177.134,6.272,148.285
C04479=1223.722,229.004,-59.276,-177.132,6.274,148.285
C04480=1223.717,229.253,-59.301,-177.129,6.276,148.285
C04481=1223.713,229.503,-59.326,-177.127,6.278,148.285
C04482=1223.708,229.751,-59.352,-177.124,6.280,148.284
C04483=1223.704,229.999,-59.378,-177.122,6.282,148.284
C04484=1223.699,230.248,-59.403,-177.119,6.284,148.284
C04485=1223.694,230.497,-59.428,-177.116,6.286,148.283
C04486=1223.690,230.746,-59.454,-177.114,6.288,148.283
C04487=1223.685,230.994,-59.479,-177.112,6.289,148.283
C04488=1223.681,231.243,-59.505,-177.109,6.291,148.282
C04489=1223.676,231.491,-59.530,-177.107,6.293,148.282
C04490=1223.672,231.740,-59.555,-177.104,6.294,148.282
C04491=1223.668,231.989,-59.581,-177.102,6.296,148.282
C04492=1223.663,232.237,-59.606,-177.099,6.298,148.281
C04493=1223.659,232.486,-59.632,-177.096,6.300,148.281
C04494=1223.654,232.735,-59.658,-177.094,6.302,148.281
C04495=1223.650,232.983,-59.683,-177.092,6.304,148.280
C04496=1223.645,233.232,-59.708,-177.089,6.306,148.280
C04497=1223.641,233.481,-59.734,-177.086,6.308,148.280
C04498=1223.636,233.729,-59.759,-177.084,6.310,148.280
C04499=1223.632,233.978,-59.785,-177.081,6.312,148.279
C04500=1223.628,234.227,-59.811,-177.078,6.313,148.279
C04501=1223.623,234.475,-59.836,-177.076,6.316,148.279
C04502=1223.618,234.724,-59.862,-177.074,6.318,148.278
C04503=1223.613,234.973,-59.888,-177.071,6.319,148.278
C04504=1223.609,235.221,-59.914,-177.068,6.321,148.278
C04505=1223.604,235.470,-59.940,-177.066,6.323,148.278
C04506=1223.600,235.719,-59.965,-177.063,6.325,148.277
C04507=1223.595,235.967,-59.991,-177.061,6.327,148.277
C04508=1223.591,236.215,-60.016,-177.058,6.329,148.277
C04509=1223.587,236.464,-60.042,-177.056,6.331,148.276
C04510=1223.583,236.713,-60.068,-177.053,6.333,148.276
C04511=1223.578,236.961,-60.093,-177.051,6.335,148.276
C04512=1223.572,237.233,-60.122,-177.048,6.337,148.276
C04513=1223.567,237.504,-60.150,-177.045,6.338,148.275
C04514=1223.563,237.776,-60.178,-177.042,6.341,148.275
C04515=1223.558,238.048,-60.206,-177.040,6.343,148.275
C04516=1223.553,238.296,-60.232,-177.037,6.345,148.274
C04517=1223.549,238.544,-60.258,-177.035,6.347,148.274
C04518=1223.545,238.793,-60.284,-177.032,6.349,148.274
C04519=1223.540,239.042,-60.310,-177.030,6.351,148.274
C04520=1223.535,239.290,-60.336,-177.027,6.353,148.273
C04521=1223.531,239.539,-60.362,-177.024,6.355,148.273
C04522=1223.527,239.788,-60.387,-177.022,6.357,148.273
C04523=1223.523,240.036,-60.413,-177.020,6.359,148.273
C04524=1223.518,240.285,-60.440,-177.017,6.360,148.272
C04525=1223.513,240.533,-60.465,-177.014,6.362,148.272
C04526=1223.509,240.782,-60.491,-177.012,6.364,148.272
C04527=1223.505,241.031,-60.517,-177.010,6.366,148.271
C04528=1223.500,241.279,-60.544,-177.007,6.368,148.271
C04529=1223.495,241.527,-60.569,-177.004,6.370,148.271
C04530=1223.491,241.776,-60.595,-177.002,6.372,148.271
C04531=1223.486,242.025,-60.622,-176.999,6.374,148.270
C04532=1223.482,242.273,-60.648,-176.997,6.376,148.270
C04533=1223.478,242.522,-60.674,-176.994,6.378,148.270
C04534=1223.473,242.771,-60.700,-176.992,6.380,148.269
C04535=1223.468,243.019,-60.726,-176.989,6.382,148.269
C04536=1223.464,243.268,-60.752,-176.987,6.384,148.269
C04537=1223.459,243.517,-60.778,-176.984,6.386,148.269
C04538=1223.455,243.765,-60.805,-176.982,6.388,148.268
C04539=1223.451,244.014,-60.830,-176.979,6.390,148.268
C04540=1223.446,244.263,-60.857,-176.977,6.391,148.268
C04541=1223.442,244.510,-60.883,-176.974,6.394,148.268
C04542=1223.437,244.759,-60.909,-176.972,6.395,148.267
C04543=1223.432,245.008,-60.935,-176.969,6.397,148.267
C04544=1223.429,245.256,-60.961,-176.967,6.399,148.267
C04545=1223.424,245.506,-60.988,-176.964,6.402,148.267
C04546=1223.420,245.754,-61.014,-176.961,6.404,148.266
C04547=1223.415,246.002,-61.040,-176.959,6.406,148.266
C04548=1223.411,246.251,-61.067,-176.956,6.408,148.266
C04549=1223.407,246.500,-61.093,-176.954,6.410,148.266
C04550=1223.401,246.748,-61.120,-176.951,6.412,148.265
C04551=1223.397,246.996,-61.145,-176.949,6.414,148.265
C04552=1223.392,247.245,-61.172,-176.946,6.416,148.265
C04553=1223.388,247.494,-61.198,-176.944,6.418,148.265
C04554=1223.384,247.742,-61.225,-176.941,6.420,148.264
C04555=1223.379,247.991,-61.251,-176.939,6.422,148.264
C04556=1223.375,248.239,-61.277,-176.936,6.423,148.264
C04557=1223.370,248.488,-61.304,-176.934,6.426,148.264
C04558=1223.366,248.736,-61.330,-176.931,6.428,148.263
C04559=1223.362,248.986,-61.357,-176.929,6.429,148.263
C04560=1223.358,249.234,-61.383,-176.927,6.432,148.263
C04561=1223.353,249.482,-61.410,-176.924,6.434,148.263
C04562=1223.349,249.731,-61.436,-176.921,6.435,148.262
C04563=1223.344,249.980,-61.463,-176.919,6.437,148.262
C04564=1223.338,250.228,-61.489,-176.916,6.440,148.262
C04565=1223.335,250.476,-61.515,-176.913,6.442,148.262
C04566=1223.330,250.725,-61.542,-176.911,6.444,148.261
C04567=1223.326,250.973,-61.568,-176.909,6.446,148.261
C04568=1223.321,251.222,-61.595,-176.906,6.448,148.261
C04569=1223.317,251.470,-61.622,-176.903,6.450,148.261
C04570=1223.312,251.719,-61.648,-176.901,6.452,148.260
C04571=1223.308,251.967,-61.674,-176.899,6.454,148.260
C04572=1223.304,252.216,-61.702,-176.896,6.456,148.260
C04573=1223.299,252.464,-61.729,-176.893,6.458,148.260
C04574=1223.295,252.713,-61.754,-176.891,6.460,148.260
C04575=1223.290,252.962,-61.781,-176.889,6.462,148.259
C04576=1223.285,253.210,-61.808,-176.886,6.464,148.259
C04577=1223.281,253.458,-61.835,-176.883,6.467,148.259
C04578=1223.276,253.708,-61.861,-176.881,6.469,148.259
C04579=1223.273,253.956,-61.888,-176.878,6.471,148.258
C04580=1223.269,254.205,-61.915,-176.876,6.473,148.258
C04581=1223.264,254.453,-61.942,-176.873,6.475,148.258
C04582=1223.260,254.702,-61.969,-176.871,6.477,148.258
C04583=1223.255,254.950,-61.996,-176.869,6.479,148.258
C04584=1223.250,255.199,-62.022,-176.866,6.481,148.257
C04585=1223.246,255.448,-62.049,-176.864,6.482,148.257
C04586=1223.242,255.696,-62.076,-176.861,6.484,148.257
C04587=1223.237,255.944,-62.103,-176.858,6.487,148.257
C04588=1223.232,256.193,-62.130,-176.856,6.489,148.256
C04589=1223.229,256.441,-62.156,-176.853,6.491,148.256
C04590=1223.224,256.690,-62.183,-176.851,6.493,148.256
C04591=1223.219,256.938,-62.210,-176.848,6.495,148.256
C04592=1223.215,257.187,-62.237,-176.846,6.497,148.256
C04593=1223.211,257.435,-62.264,-176.844,6.499,148.255
C04594=1223.206,257.683,-62.291,-176.841,6.501,148.255
C04595=1223.202,257.932,-62.318,-176.839,6.503,148.255
C04596=1223.197,258.181,-62.345,-176.836,6.506,148.255
C04597=1223.193,258.429,-62.372,-176.833,6.508,148.254
C04598=1223.189,258.678,-62.399,-176.831,6.510,148.254
C04599=1223.184,258.926,-62.426,-176.828,6.512,148.254
C04600=1223.179,259.175,-62.453,-176.826,6.514,148.254
C04601=1223.175,259.423,-62.480,-176.824,6.516,148.253
C04602=1223.171,259.671,-62.507,-176.821,6.518,148.253
C04603=1223.167,259.920,-62.534,-176.819,6.520,148.253
C04604=1223.162,260.169,-62.561,-176.816,6.523,148.253
C04605=1223.157,260.417,-62.588,-176.813,6.525,148.253
C04606=1223.153,260.666,-62.615,-176.811,6.527,148.252
C04607=1223.148,260.914,-62.642,-176.808,6.529,148.252
C04608=1223.144,261.163,-62.669,-176.806,6.531,148.252
C04609=1223.140,261.411,-62.697,-176.804,6.533,148.252
C04610=1223.136,261.660,-62.724,-176.801,6.535,148.251
C04611=1223.131,261.908,-62.751,-176.799,6.537,148.251
C04612=1223.126,262.157,-62.778,-176.796,6.540,148.251
C04613=1223.122,262.405,-62.805,-176.793,6.542,148.251
C04614=1223.117,262.654,-62.832,-176.791,6.544,148.251
C04615=1223.113,262.902,-62.860,-176.788,6.546,148.250
C04616=1223.109,263.175,-62.889,-176.786,6.548,148.250
C04617=1223.103,263.448,-62.920,-176.783,6.551,148.250
C04618=1223.099,263.720,-62.949,-176.780,6.553,148.250
C04619=1223.094,263.993,-62.980,-176.777,6.555,148.250
C04620=1223.089,264.241,-63.007,-176.775,6.557,148.249
C04621=1223.085,264.489,-63.034,-176.773,6.559,148.249
C04622=1223.081,264.738,-63.061,-176.770,6.561,148.249
C04623=1223.077,264.987,-63.088,-176.768,6.563,148.249
C04624=1223.072,265.235,-63.116,-176.765,6.566,148.249
C04625=1223.068,265.483,-63.143,-176.763,6.568,148.248
C04626=1223.063,265.732,-63.171,-176.760,6.570,148.248
C04627=1223.059,265.981,-63.198,-176.758,6.572,148.248
C04628=1223.054,266.228,-63.226,-176.755,6.574,148.248
C04629=1223.050,266.477,-63.253,-176.753,6.576,148.247
C04630=1223.045,266.726,-63.281,-176.750,6.579,148.247
C04631=1223.041,266.974,-63.308,-176.747,6.581,148.247
C04632=1223.036,267.223,-63.335,-176.745,6.583,148.247
C04633=1223.032,267.471,-63.363,-176.743,6.585,148.247
C04634=1223.028,267.720,-63.391,-176.740,6.587,148.247
C04635=1223.023,267.968,-63.418,-176.737,6.590,148.246
C04636=1223.019,268.216,-63.446,-176.735,6.592,148.246
C04637=1223.015,268.465,-63.474,-176.733,6.594,148.246
C04638=1223.010,268.713,-63.501,-176.730,6.596,148.246
C04639=1223.006,268.961,-63.528,-176.728,6.598,148.246
C04640=1223.001,269.210,-63.556,-176.725,6.600,148.245
C04641=1222.997,269.458,-63.584,-176.723,6.603,148.245
C04642=1222.993,269.707,-63.611,-176.720,6.605,148.245
C04643=1222.988,269.955,-63.639,-176.718,6.607,148.245
C04644=1222.984,270.204,-63.667,-176.715,6.609,148.245
C04645=1222.979,270.452,-63.694,-176.713,6.611,148.245
C04646=1222.975,270.701,-63.721,-176.710,6.614,148.244
C04647=1222.971,270.949,-63.750,-176.708,6.616,148.244
C04648=1222.966,271.198,-63.777,-176.705,6.618,148.244
C04649=1222.961,271.446,-63.805,-176.703,6.620,148.244
C04650=1222.957,271.694,-63.833,-176.701,6.622,148.244
C04651=1222.953,271.943,-63.860,-176.698,6.625,148.244
C04652=1222.948,272.191,-63.888,-176.695,6.627,148.243
C04653=1222.944,272.440,-63.915,-176.693,6.630,148.243
C04654=1222.939,272.688,-63.944,-176.691,6.631,148.243
C04655=1222.935,272.937,-63.972,-176.688,6.634,148.243
C04656=1222.931,273.185,-63.999,-176.685,6.636,148.243
C04657=1222.926,273.433,-64.027,-176.683,6.639,148.243
C04658=1222.923,273.682,-64.055,-176.681,6.640,148.242
C04659=1222.918,273.930,-64.083,-176.678,6.643,148.242
C04660=1222.914,274.179,-64.111,-176.676,6.645,148.242
C04661=1222.909,274.427,-64.138,-176.673,6.648,148.242
C04662=1222.905,274.675,-64.166,-176.671,6.649,148.242
C04663=1222.900,274.924,-64.195,-176.668,6.652,148.242
C04664=1222.896,275.172,-64.222,-176.666,6.654,148.241
C04665=1222.892,275.421,-64.250,-176.663,6.657,148.241
C04666=1222.887,275.669,-64.279,-176.661,6.658,148.241
C04667=1222.883,275.917,-64.306,-176.658,6.661,148.241
C04668=1222.879,276.165,-64.334,-176.656,6.663,148.241
C04669=1222.873,276.414,-64.362,-176.654,6.665,148.240
C04670=1222.870,276.663,-64.390,-176.651,6.668,148.240
C04671=1222.865,276.911,-64.418,-176.648,6.670,148.240
C04672=1222.861,277.160,-64.447,-176.646,6.672,148.240
C04673=1222.856,277.407,-64.475,-176.644,6.674,148.240
C04674=1222.853,277.656,-64.503,-176.641,6.677,148.240
C04675=1222.848,277.904,-64.531,-176.638,6.679,148.239
C04676=1222.844,278.153,-64.558,-176.636,6.681,148.239
C04677=1222.839,278.401,-64.586,-176.634,6.683,148.239
C04678=1222.834,278.649,-64.615,-176.631,6.686,148.239
C04679=1222.830,278.898,-64.643,-176.629,6.688,148.239
C04680=1222.825,279.146,-64.671,-176.626,6.690,148.239
C04681=1222.822,279.395,-64.699,-176.624,6.692,148.239
C04682=1222.817,279.643,-64.727,-176.621,6.695,148.238
C04683=1222.813,279.892,-64.756,-176.619,6.697,148.238
C04684=1222.808,280.139,-64.784,-176.617,6.699,148.238
C04685=1222.804,280.388,-64.812,-176.614,6.701,148.238
C04686=1222.800,280.636,-64.840,-176.612,6.704,148.238
C04687=1222.795,280.885,-64.869,-176.609,6.706,148.238
C04688=1222.791,281.134,-64.897,-176.607,6.708,148.238
C04689=1222.787,281.382,-64.925,-176.605,6.711,148.238
C04690=1222.782,281.630,-64.954,-176.602,6.713,148.237
C04691=1222.778,281.878,-64.981,-176.599,6.715,148.237
C04692=1222.774,282.127,-65.011,-176.597,6.717,148.237
C04693=1222.770,282.374,-65.039,-176.595,6.720,148.237
C04694=1222.765,282.623,-65.067,-176.592,6.723,148.237
C04695=1222.761,282.871,-65.095,-176.589,6.725,148.237
C04696=1222.756,283.120,-65.124,-176.587,6.727,148.236
C04697=1222.752,283.368,-65.152,-176.585,6.730,148.236
C04698=1222.747,283.617,-65.180,-176.582,6.732,148.236
C04699=1222.743,283.866,-65.209,-176.580,6.734,148.236
C04700=1222.739,284.113,-65.238,-176.577,6.736,148.236
C04701=1222.734,284.362,-65.266,-176.575,6.739,148.236
C04702=1222.730,284.610,-65.294,-176.573,6.741,148.236
C04703=1222.726,284.859,-65.323,-176.570,6.743,148.235
C04704=1222.721,285.106,-65.351,-176.568,6.745,148.235
C04705=1222.717,285.355,-65.380,-176.565,6.748,148.235
C04706=1222.713,285.604,-65.409,-176.563,6.750,148.235
C04707=1222.708,285.852,-65.437,-176.560,6.752,148.235
C04708=1222.704,286.100,-65.466,-176.558,6.755,148.235
C04709=1222.700,286.349,-65.495,-176.555,6.757,148.235
C04710=1222.695,286.597,-65.522,-176.553,6.759,148.235
C04711=1222.691,286.845,-65.551,-176.551,6.762,148.235
C04712=1222.687,287.093,-65.580,-176.548,6.764,148.234
C04713=1222.682,287.342,-65.608,-176.546,6.767,148.234
C04714=1222.678,287.590,-65.637,-176.544,6.769,148.234
C04715=1222.674,287.838,-65.666,-176.540,6.772,148.234
C04716=1222.669,288.087,-65.694,-176.538,6.774,148.234
C04717=1222.665,288.335,-65.724,-176.536,6.776,148.234
C04718=1222.661,288.583,-65.752,-176.534,6.778,148.234
C04719=1222.656,288.832,-65.780,-176.531,6.781,148.234
C04720=1222.652,289.105,-65.813,-176.529,6.783,148.233
C04721=1222.647,289.380,-65.844,-176.526,6.786,148.233
C04722=1222.642,289.654,-65.876,-176.523,6.789,148.233
C04723=1222.637,289.928,-65.907,-176.521,6.791,148.233
C04724=1222.632,290.176,-65.937,-176.518,6.794,148.233
C04725=1222.628,290.425,-65.965,-176.516,6.796,148.233
C04726=1222.624,290.673,-65.994,-176.514,6.798,148.233
C04727=1222.619,290.921,-66.023,-176.511,6.801,148.233
C04728=1222.615,291.169,-66.052,-176.508,6.803,148.232
C04729=1222.611,291.418,-66.081,-176.506,6.805,148.232
C04730=1222.607,291.665,-66.109,-176.503,6.808,148.232
C04731=1222.602,291.914,-66.138,-176.501,6.811,148.232
C04732=1222.598,292.163,-66.168,-176.499,6.813,148.232
C04733=1222.594,292.412,-66.196,-176.497,6.815,148.232
C04734=1222.589,292.659,-66.225,-176.494,6.818,148.232
C04735=1222.585,292.907,-66.254,-176.492,6.820,148.232
C04736=1222.581,293.156,-66.283,-176.489,6.822,148.232
C04737=1222.577,293.404,-66.312,-176.487,6.825,148.232
C04738=1222.572,293.652,-66.341,-176.484,6.827,148.232
C04739=1222.567,293.901,-66.370,-176.482,6.829,148.232
C04740=1222.563,294.149,-66.400,-176.479,6.832,148.231
C04741=1222.559,294.397,-66.428,-176.477,6.834,148.231
C04742=1222.555,294.645,-66.457,-176.475,6.837,148.231
C04743=1222.550,294.893,-66.486,-176.472,6.840,148.231
C04744=1222.546,295.142,-66.515,-176.470,6.842,148.231
C04745=1222.542,295.390,-66.545,-176.468,6.844,148.231
C04746=1222.537,295.638,-66.574,-176.465,6.847,148.231
C04747=1222.533,295.886,-66.603,-176.463,6.849,148.231
C04748=1222.528,296.135,-66.632,-176.461,6.851,148.231
C04749=1222.524,296.383,-66.661,-176.458,6.854,148.231
C04750=1222.520,296.632,-66.691,-176.455,6.856,148.230
C04751=1222.516,296.880,-66.720,-176.453,6.858,148.230
C04752=1222.511,297.128,-66.748,-176.451,6.861,148.230
C04753=1222.507,297.376,-66.777,-176.449,6.864,148.230
C04754=1222.503,297.624,-66.807,-176.446,6.866,148.230
C04755=1222.499,297.873,-66.836,-176.444,6.869,148.230
C04756=1222.495,298.121,-66.866,-176.441,6.871,148.230
C04757=1222.491,298.369,-66.895,-176.439,6.873,148.230
C04758=1222.485,298.617,-66.924,-176.436,6.876,148.230
C04759=1222.481,298.866,-66.953,-176.434,6.878,148.230
C04760=1222.477,299.114,-66.983,-176.432,6.880,148.230
C04761=1222.473,299.362,-67.012,-176.430,6.883,148.230
C04762=1222.469,299.610,-67.041,-176.427,6.886,148.230
C04763=1222.465,299.859,-67.071,-176.424,6.888,148.229
C04764=1222.460,300.106,-67.100,-176.422,6.891,148.229
C04765=1222.456,300.355,-67.129,-176.420,6.893,148.229
C04766=1222.451,300.603,-67.160,-176.417,6.896,148.229
C04767=1222.446,300.851,-67.189,-176.415,6.898,148.229
C04768=1222.442,301.100,-67.218,-176.413,6.900,148.229
C04769=1222.438,301.348,-67.248,-176.411,6.903,148.229
C04770=1222.434,301.596,-67.277,-176.408,6.906,148.229
C04771=1222.430,301.844,-67.307,-176.406,6.908,148.229
C04772=1222.426,302.093,-67.336,-176.403,6.911,148.229
C04773=1222.421,302.341,-67.366,-176.401,6.913,148.229
C04774=1222.417,302.589,-67.395,-176.399,6.915,148.229
C04775=1222.412,302.837,-67.424,-176.396,6.918,148.229
C04776=1222.408,303.085,-67.454,-176.394,6.920,148.229
C04777=1222.403,303.334,-67.484,-176.391,6.923,148.229
C04778=1222.399,303.582,-67.513,-176.389,6.925,148.229
C04779=1222.395,303.830,-67.543,-176.387,6.928,148.229
C04780=1222.391,304.078,-67.572,-176.385,6.931,148.229
C04781=1222.387,304.327,-67.602,-176.382,6.933,148.228
C04782=1222.383,304.574,-67.632,-176.380,6.935,148.228
C04783=1222.378,304.823,-67.662,-176.378,6.938,148.228
C04784=1222.374,305.071,-67.691,-176.376,6.940,148.228
C04785=1222.369,305.320,-67.721,-176.373,6.943,148.228
C04786=1222.365,305.568,-67.750,-176.371,6.946,148.228
C04787=1222.361,305.816,-67.780,-176.369,6.948,148.228
C04788=1222.356,306.064,-67.810,-176.366,6.951,148.228
C04789=1222.352,306.312,-67.840,-176.364,6.953,148.228
C04790=1222.348,306.561,-67.869,-176.362,6.955,148.228
C04791=1222.344,306.809,-67.899,-176.359,6.958,148.228
C04792=1222.339,307.057,-67.929,-176.357,6.961,148.228
C04793=1222.335,307.305,-67.959,-176.355,6.963,148.228
C04794=1222.331,307.553,-67.988,-176.352,6.966,148.228
C04795=1222.327,307.802,-68.018,-176.350,6.968,148.228
C04796=1222.322,308.050,-68.049,-176.347,6.971,148.228
C04797=1222.318,308.298,-68.078,-176.345,6.973,148.228
C04798=1222.314,308.546,-68.107,-176.343,6.976,148.228
C04799=1222.309,308.794,-68.138,-176.341,6.979,148.228
C04800=1222.305,309.042,-68.168,-176.339,6.981,148.228
C04801=1222.301,309.291,-68.197,-176.336,6.983,148.228
C04802=1222.296,309.539,-68.228,-176.334,6.986,148.228
C04803=1222.292,309.787,-68.257,-176.332,6.988,148.228
C04804=1222.288,310.035,-68.287,-176.329,6.991,148.228
C04805=1222.283,310.283,-68.318,-176.327,6.994,148.228
C04806=1222.279,310.531,-68.347,-176.325,6.996,148.228
C04807=1222.275,310.779,-68.377,-176.322,6.999,148.228
C04808=1222.270,311.028,-68.407,-176.320,7.001,148.227
C04809=1222.266,311.275,-68.437,-176.317,7.004,148.227
C04810=1222.261,311.524,-68.467,-176.315,7.006,148.227
C04811=1222.258,311.771,-68.498,-176.313,7.009,148.227
C04812=1222.253,312.020,-68.527,-176.310,7.012,148.227
C04813=1222.249,312.268,-68.558,-176.309,7.014,148.228
C04814=1222.245,312.517,-68.588,-176.306,7.017,148.228
C04815=1222.241,312.765,-68.618,-176.304,7.019,148.227
C04816=1222.236,313.013,-68.648,-176.302,7.022,148.227
C04817=1222.233,313.260,-68.678,-176.299,7.025,148.227
C04818=1222.228,313.509,-68.708,-176.297,7.027,148.227
C04819=1222.224,313.757,-68.738,-176.295,7.029,148.227
C04820=1222.219,314.005,-68.768,-176.292,7.032,148.227
C04821=1222.215,314.253,-68.799,-176.291,7.035,148.227
C04822=1222.210,314.501,-68.829,-176.288,7.038,148.227
C04823=1222.207,314.750,-68.859,-176.286,7.040,148.227
C04824=1222.201,315.025,-68.893,-176.283,7.043,148.227
C04825=1222.197,315.301,-68.926,-176.281,7.046,148.227
C04826=1222.192,315.577,-68.960,-176.279,7.048,148.227
C04827=1222.187,315.853,-68.994,-176.276,7.051,148.227
C04828=1222.183,316.101,-69.024,-176.273,7.054,148.227
C04829=1222.179,316.349,-69.055,-176.271,7.057,148.227
C04830=1222.174,316.597,-69.084,-176.269,7.059,148.228
C04831=1222.170,316.846,-69.115,-176.267,7.062,148.228
C04832=1222.167,317.093,-69.146,-176.265,7.064,148.227
C04833=1222.162,317.342,-69.176,-176.262,7.067,148.227
C04834=1222.158,317.590,-69.206,-176.260,7.070,148.227
C04835=1222.153,317.838,-69.236,-176.258,7.072,148.228
C04836=1222.149,318.086,-69.268,-176.256,7.075,148.228
C04837=1222.145,318.334,-69.297,-176.254,7.077,148.228
C04838=1222.140,318.582,-69.328,-176.251,7.081,148.228
C04839=1222.136,318.830,-69.358,-176.249,7.083,148.228
C04840=1222.132,319.078,-69.389,-176.247,7.085,148.228
C04841=1222.128,319.327,-69.420,-176.244,7.088,148.228
C04842=1222.124,319.574,-69.450,-176.242,7.091,148.228
C04843=1222.119,319.823,-69.480,-176.240,7.094,148.228
C04844=1222.115,320.071,-69.510,-176.238,7.096,148.228
C04845=1222.111,320.319,-69.541,-176.236,7.098,148.228
C04846=1222.107,320.567,-69.572,-176.233,7.101,148.228
C04847=1222.103,320.815,-69.602,-176.231,7.104,148.228
C04848=1222.098,321.063,-69.633,-176.229,7.107,148.228
C04849=1222.093,321.311,-69.664,-176.227,7.109,148.228
C04850=1222.090,321.559,-69.694,-176.225,7.111,148.228
C04851=1222.086,321.807,-69.725,-176.223,7.115,148.228
C04852=1222.081,322.055,-69.756,-176.221,7.117,148.228
C04853=1222.077,322.304,-69.786,-176.218,7.120,148.228
C04854=1222.073,322.552,-69.817,-176.216,7.122,148.228
C04855=1222.068,322.800,-69.847,-176.214,7.125,148.228
C04856=1222.064,323.048,-69.878,-176.211,7.128,148.228
C04857=1222.060,323.296,-69.909,-176.209,7.130,148.228
C04858=1222.056,323.544,-69.939,-176.207,7.133,148.228
C04859=1222.051,323.792,-69.971,-176.205,7.136,148.228
C04860=1222.047,324.040,-70.002,-176.203,7.138,148.228
C04861=1222.043,324.288,-70.032,-176.201,7.141,148.228
C04862=1222.039,324.536,-70.063,-176.199,7.143,148.228
C04863=1222.034,324.784,-70.094,-176.196,7.147,148.229
C04864=1222.030,325.032,-70.125,-176.194,7.149,148.229
C04865=1222.026,325.280,-70.155,-176.192,7.151,148.229
C04866=1222.022,325.528,-70.186,-176.190,7.155,148.229
C04867=1222.018,325.777,-70.217,-176.188,7.157,148.229
C04868=1222.013,326.025,-70.248,-176.185,7.160,148.229
C04869=1222.008,326.273,-70.278,-176.184,7.162,148.229
C04870=1222.005,326.521,-70.310,-176.182,7.165,148.229
C04871=1222.001,326.768,-70.340,-176.179,7.168,148.229
C04872=1221.997,327.017,-70.372,-176.177,7.170,148.229
C04873=1221.992,327.265,-70.402,-176.175,7.173,148.229
C04874=1221.988,327.513,-70.433,-176.173,7.176,148.229
C04875=1221.984,327.761,-70.465,-176.171,7.178,148.229
C04876=1221.979,328.009,-70.496,-176.169,7.181,148.229
C04877=1221.975,328.257,-70.526,-176.167,7.184,148.229
C04878=1221.971,328.505,-70.557,-176.164,7.187,148.230
C04879=1221.967,328.752,-70.588,-176.162,7.189,148.230
C04880=1221.963,329.001,-70.620,-176.161,7.192,148.230
C04881=1221.959,329.249,-70.650,-176.158,7.195,148.230
C04882=1221.954,329.497,-70.681,-176.156,7.197,148.230
C04883=1221.950,329.745,-70.713,-176.154,7.200,148.230
C04884=1221.946,329.993,-70.744,-176.152,7.203,148.230
C04885=1221.941,330.241,-70.774,-176.150,7.205,148.230
C04886=1221.937,330.489,-70.806,-176.147,7.208,148.230
C04887=1221.933,330.737,-70.837,-176.146,7.211,148.230
C04888=1221.929,330.986,-70.868,-176.143,7.214,148.230
C04889=1221.924,331.233,-70.900,-176.141,7.216,148.230
C04890=1221.920,331.482,-70.931,-176.139,7.218,148.230
C04891=1221.916,331.729,-70.962,-176.137,7.222,148.231
C04892=1221.911,331.977,-70.993,-176.135,7.224,148.231
C04893=1221.907,332.226,-71.024,-176.133,7.227,148.231
C04894=1221.903,332.473,-71.056,-176.131,7.230,148.231
C04895=1221.899,332.722,-71.087,-176.129,7.232,148.231
C04896=1221.895,332.969,-71.118,-176.127,7.235,148.231
C04897=1221.891,333.218,-71.149,-176.125,7.238,148.231
C04898=1221.886,333.465,-71.181,-176.123,7.241,148.231
C04899=1221.882,333.714,-71.212,-176.120,7.243,148.231
C04900=1221.878,333.961,-71.243,-176.119,7.246,148.231
C04901=1221.874,334.210,-71.275,-176.117,7.249,148.232
C04902=1221.870,334.457,-71.306,-176.115,7.251,148.232
C04903=1221.866,334.706,-71.337,-176.112,7.255,148.232
C04904=1221.862,334.953,-71.369,-176.110,7.257,148.232
C04905=1221.857,335.202,-71.400,-176.109,7.259,148.232
C04906=1221.853,335.449,-71.431,-176.106,7.263,148.232
C04907=1221.849,335.698,-71.462,-176.104,7.265,148.232
C04908=1221.845,335.945,-71.494,-176.102,7.268,148.232
C04909=1221.840,336.193,-71.526,-176.101,7.271,148.233
C04910=1221.836,336.441,-71.557,-176.098,7.273,148.233
C04911=1221.832,336.689,-71.589,-176.096,7.277,148.233
C04912=1221.827,336.937,-71.620,-176.094,7.279,148.233
C04913=1221.824,337.185,-71.652,-176.092,7.282,148.233
C04914=1221.819,337.433,-71.683,-176.090,7.285,148.233
C04915=1221.815,337.681,-71.714,-176.088,7.287,148.233
C04916=1221.810,337.929,-71.746,-176.086,7.290,148.233
C04917=1221.807,338.177,-71.778,-176.084,7.293,148.233
C04918=1221.802,338.425,-71.809,-176.083,7.295,148.234
C04919=1221.798,338.673,-71.841,-176.080,7.298,148.234
C04920=1221.794,338.920,-71.872,-176.078,7.301,148.234
C04921=1221.790,339.168,-71.904,-176.076,7.304,148.234
C04922=1221.786,339.417,-71.936,-176.074,7.306,148.234
C04923=1221.781,339.665,-71.967,-176.073,7.309,148.234
C04924=1221.778,339.913,-71.999,-176.070,7.312,148.234
C04925=1221.773,340.160,-72.031,-176.069,7.315,148.235
C04926=1221.769,340.409,-72.062,-176.067,7.317,148.235
C04927=1221.764,340.656,-72.094,-176.064,7.320,148.235
C04928=1221.760,340.934,-72.129,-176.062,7.324,148.235
C04929=1221.755,341.212,-72.164,-176.061,7.326,148.235
C04930=1221.750,341.490,-72.200,-176.058,7.329,148.235
C04931=1221.746,341.767,-72.236,-176.056,7.333,148.235
C04932=1221.742,342.015,-72.268,-176.054,7.335,148.236
C04933=1221.737,342.263,-72.300,-176.052,7.339,148.236
C04934=1221.733,342.512,-72.331,-176.050,7.341,148.236
C04935=1221.729,342.760,-72.363,-176.048,7.343,148.236
C04936=1221.724,343.007,-72.395,-176.046,7.347,148.236
C04937=1221.721,343.255,-72.427,-176.044,7.349,148.236
C04938=1221.716,343.503,-72.458,-176.042,7.353,148.237
C04939=1221.712,343.751,-72.491,-176.041,7.355,148.237
C04940=1221.708,343.999,-72.523,-176.039,7.358,148.237
C04941=1221.704,344.247,-72.554,-176.037,7.361,148.237
C04942=1221.699,344.495,-72.587,-176.035,7.363,148.237
C04943=1221.696,344.743,-72.618,-176.033,7.366,148.237
C04944=1221.691,344.990,-72.650,-176.031,7.369,148.238
C04945=1221.687,345.239,-72.682,-176.029,7.372,148.238
C04946=1221.683,345.487,-72.714,-176.028,7.374,148.238
C04947=1221.678,345.734,-72.746,-176.025,7.378,148.238
C04948=1221.675,345.982,-72.778,-176.024,7.380,148.238
C04949=1221.671,346.230,-72.810,-176.022,7.383,148.239
C04950=1221.666,346.478,-72.842,-176.020,7.386,148.239
C04951=1221.662,346.726,-72.874,-176.018,7.388,148.239
C04952=1221.658,346.974,-72.906,-176.016,7.391,148.239
C04953=1221.653,347.222,-72.938,-176.014,7.394,148.239
C04954=1221.650,347.470,-72.970,-176.012,7.397,148.239
C04955=1221.645,347.718,-73.002,-176.010,7.400,148.240
C04956=1221.641,347.965,-73.034,-176.009,7.402,148.240
C04957=1221.636,348.214,-73.066,-176.007,7.405,148.240
C04958=1221.633,348.461,-73.099,-176.005,7.408,148.240
C04959=1221.629,348.710,-73.131,-176.003,7.411,148.240
C04960=1221.624,348.957,-73.162,-176.001,7.413,148.241
C04961=1221.620,349.205,-73.195,-175.999,7.417,148.241
C04962=1221.616,349.453,-73.227,-175.998,7.419,148.241
C04963=1221.611,349.701,-73.259,-175.996,7.422,148.241
C04964=1221.608,349.948,-73.291,-175.994,7.425,148.241
C04965=1221.603,350.197,-73.324,-175.992,7.428,148.242
C04966=1221.600,350.445,-73.356,-175.990,7.430,148.242
C04967=1221.595,350.692,-73.388,-175.989,7.434,148.242
C04968=1221.591,350.940,-73.420,-175.987,7.436,148.242
C04969=1221.587,351.188,-73.453,-175.985,7.439,148.243
C04970=1221.583,351.436,-73.485,-175.984,7.441,148.243
C04971=1221.578,351.684,-73.517,-175.982,7.445,148.243
C04972=1221.575,351.931,-73.549,-175.980,7.447,148.243
C04973=1221.570,352.180,-73.582,-175.978,7.450,148.243
C04974=1221.566,352.428,-73.614,-175.976,7.453,148.244
C04975=1221.562,352.675,-73.647,-175.975,7.456,148.244
C04976=1221.557,352.923,-73.679,-175.973,7.458,148.244
C04977=1221.553,353.171,-73.711,-175.971,7.462,148.244
C04978=1221.549,353.419,-73.744,-175.970,7.464,148.245
C04979=1221.546,353.667,-73.776,-175.968,7.467,148.245
C04980=1221.541,353.914,-73.808,-175.966,7.470,148.245
C04981=1221.536,354.162,-73.841,-175.964,7.473,148.245
C04982=1221.533,354.410,-73.873,-175.962,7.475,148.245
C04983=1221.528,354.659,-73.905,-175.961,7.478,148.246
C04984=1221.524,354.906,-73.938,-175.959,7.482,148.246
C04985=1221.520,355.154,-73.970,-175.957,7.484,148.246
C04986=1221.516,355.401,-74.003,-175.956,7.487,148.246
C04987=1221.511,355.650,-74.035,-175.954,7.490,148.247
C04988=1221.508,355.897,-74.068,-175.952,7.493,148.247
C04989=1221.503,356.146,-74.100,-175.951,7.495,148.247
C04990=1221.500,356.393,-74.133,-175.949,7.498,148.247
C04991=1221.496,356.641,-74.165,-175.947,7.501,148.248
C04992=1221.491,356.889,-74.197,-175.945,7.504,148.248
C04993=1221.486,357.137,-74.231,-175.944,7.506,148.248
C04994=1221.483,357.384,-74.263,-175.942,7.510,148.248
C04995=1221.479,357.632,-74.296,-175.940,7.512,148.249
C04996=1221.474,357.880,-74.329,-175.939,7.515,148.249
C04997=1221.471,358.128,-74.361,-175.938,7.518,148.249
C04998=1221.467,358.376,-74.394,-175.935,7.521,148.249
C04999=1221.462,358.624,-74.426,-175.934,7.524,148.250
C05000=1221.457,358.871,-74.459,-175.933,7.526,148.250
C05001=1221.454,359.119,-74.491,-175.931,7.529,148.250
C05002=1221.450,359.367,-74.524,-175.929,7.532,148.250
C05003=1221.445,359.615,-74.557,-175.928,7.535,148.251
C05004=1221.441,359.863,-74.590,-175.926,7.538,148.251
C05005=1221.438,360.111,-74.622,-175.925,7.540,148.251
C05006=1221.433,360.359,-74.655,-175.923,7.544,148.252
C05007=1221.429,360.607,-74.688,-175.921,7.546,148.252
C05008=1221.425,360.854,-74.721,-175.920,7.549,148.252
C05009=1221.421,361.102,-74.752,-175.918,7.552,148.252
C05010=1221.416,361.349,-74.786,-175.916,7.555,148.253
C05011=1221.412,361.597,-74.819,-175.915,7.558,148.253
C05012=1221.408,361.846,-74.851,-175.913,7.560,148.253
C05013=1221.404,362.093,-74.884,-175.912,7.563,148.254
C05014=1221.400,362.341,-74.917,-175.910,7.567,148.254
C05015=1221.396,362.588,-74.950,-175.909,7.569,148.254
C05016=1221.392,362.837,-74.982,-175.907,7.572,148.254
C05017=1221.388,363.084,-75.016,-175.906,7.575,148.255
C05018=1221.383,363.332,-75.049,-175.904,7.577,148.255
C05019=1221.379,363.580,-75.082,-175.902,7.581,148.255
C05020=1221.375,363.828,-75.114,-175.901,7.583,148.256
C05021=1221.371,364.076,-75.147,-175.900,7.586,148.256
C05022=1221.367,364.323,-75.180,-175.898,7.589,148.256
C05023=1221.363,364.571,-75.213,-175.897,7.592,148.257
C05024=1221.359,364.819,-75.246,-175.895,7.594,148.257
C05025=1221.355,365.067,-75.279,-175.893,7.598,148.257
C05026=1221.350,365.315,-75.312,-175.892,7.600,148.257
C05027=1221.346,365.563,-75.345,-175.891,7.603,148.258
C05028=1221.342,365.810,-75.378,-175.889,7.606,148.258
C05029=1221.339,366.058,-75.411,-175.888,7.608,148.258
C05030=1221.335,366.306,-75.444,-175.887,7.611,148.259
C05031=1221.331,366.553,-75.477,-175.884,7.615,148.259
C05032=1221.326,366.834,-75.514,-175.883,7.618,148.259
C05033=1221.321,367.113,-75.551,-175.882,7.621,148.260
C05034=1221.316,367.393,-75.589,-175.880,7.624,148.260
C05035=1221.311,367.673,-75.626,-175.878,7.627,148.260
C05036=1221.307,367.921,-75.659,-175.877,7.630,148.261
C05037=1221.303,368.168,-75.692,-175.875,7.633,148.261
C05038=1221.299,368.416,-75.725,-175.874,7.636,148.261
C05039=1221.295,368.664,-75.758,-175.873,7.638,148.262
C05040=1221.291,368.912,-75.792,-175.871,7.641,148.262
C05041=1221.287,369.159,-75.825,-175.870,7.644,148.262
C05042=1221.283,369.407,-75.858,-175.868,7.647,148.263
C05043=1221.278,369.655,-75.891,-175.867,7.650,148.263
C05044=1221.274,369.902,-75.924,-175.866,7.653,148.263
C05045=1221.270,370.150,-75.957,-175.864,7.655,148.264
C05046=1221.266,370.398,-75.991,-175.863,7.658,148.264
C05047=1221.262,370.646,-76.024,-175.862,7.661,148.264
C05048=1221.258,370.893,-76.057,-175.860,7.664,148.265
C05049=1221.254,371.141,-76.090,-175.859,7.666,148.265
C05050=1221.249,371.389,-76.123,-175.858,7.669,148.266
C05051=1221.245,371.637,-76.156,-175.856,7.672,148.266
C05052=1221.241,371.885,-76.191,-175.855,7.675,148.266
C05053=1221.237,372.132,-76.224,-175.854,7.677,148.267
C05054=1221.233,372.380,-76.257,-175.853,7.680,148.267
C05055=1221.229,372.628,-76.291,-175.852,7.683,148.267
C05056=1221.225,372.876,-76.324,-175.850,7.686,148.268
C05057=1221.221,373.123,-76.357,-175.849,7.688,148.268
C05058=1221.216,373.371,-76.390,-175.848,7.691,148.268
C05059=1221.212,373.619,-76.423,-175.847,7.694,148.269
C05060=1221.209,373.866,-76.457,-175.845,7.697,148.269
C05061=1221.204,374.114,-76.490,-175.844,7.700,148.270
C05062=1221.200,374.361,-76.523,-175.843,7.703,148.270
C05063=1221.196,374.610,-76.558,-175.841,7.705,148.270
C05064=1221.192,374.858,-76.591,-175.840,7.708,148.271
C05065=1221.188,375.106,-76.624,-175.839,7.711,148.271
C05066=1221.184,375.353,-76.658,-175.838,7.714,148.271
C05067=1221.180,375.600,-76.691,-175.837,7.716,148.272
C05068=1221.176,375.848,-76.724,-175.836,7.719,148.272
C05069=1221.171,376.096,-76.757,-175.834,7.722,148.272
C05070=1221.167,376.343,-76.792,-175.833,7.725,148.273
C05071=1221.163,376.591,-76.825,-175.832,7.728,148.273
C05072=1221.159,376.839,-76.858,-175.831,7.730,148.274
C05073=1221.155,377.087,-76.892,-175.830,7.733,148.274
C05074=1221.151,377.334,-76.925,-175.828,7.736,148.274
C05075=1221.147,377.582,-76.959,-175.827,7.739,148.275
C05076=1221.142,377.830,-76.992,-175.826,7.742,148.275
C05077=1221.138,378.078,-77.025,-175.825,7.744,148.276
C05078=1221.134,378.325,-77.059,-175.824,7.747,148.276
C05079=1221.131,378.573,-77.093,-175.823,7.749,148.276
C05080=1221.127,378.821,-77.126,-175.822,7.752,148.277
C05081=1221.122,379.068,-77.160,-175.821,7.755,148.277
C05082=1221.118,379.316,-77.194,-175.820,7.758,148.278
C05083=1221.114,379.564,-77.227,-175.818,7.761,148.278
C05084=1221.110,379.811,-77.261,-175.817,7.763,148.278
C05085=1221.106,380.060,-77.295,-175.817,7.765,148.279
C05086=1221.102,380.307,-77.329,-175.815,7.768,148.279
C05087=1221.098,380.555,-77.362,-175.814,7.771,148.280
C05088=1221.094,380.802,-77.395,-175.813,7.774,148.280
C05089=1221.089,381.050,-77.429,-175.812,7.777,148.280
C05090=1221.085,381.297,-77.463,-175.811,7.779,148.281
C05091=1221.082,381.545,-77.497,-175.810,7.781,148.281
C05092=1221.077,381.793,-77.530,-175.809,7.784,148.281
C05093=1221.073,382.041,-77.564,-175.808,7.787,148.282
C05094=1221.069,382.288,-77.598,-175.807,7.790,148.282
C05095=1221.065,382.536,-77.631,-175.806,7.793,148.283
C05096=1221.061,382.784,-77.666,-175.805,7.795,148.283
C05097=1221.056,383.032,-77.699,-175.804,7.798,148.284
C05098=1221.053,383.279,-77.733,-175.803,7.801,148.284
C05099=1221.048,383.527,-77.766,-175.802,7.803,148.284
C05100=1221.044,383.774,-77.800,-175.800,7.806,148.285
C05101=1221.040,384.022,-77.834,-175.800,7.809,148.285
C05102=1221.036,384.270,-77.868,-175.799,7.811,148.286
C05103=1221.032,384.518,-77.901,-175.798,7.814,148.286
C05104=1221.028,384.765,-77.935,-175.797,7.817,148.286
C05105=1221.024,385.013,-77.969,-175.796,7.819,148.287
C05106=1221.020,385.261,-78.003,-175.795,7.822,148.287
C05107=1221.016,385.508,-78.036,-175.794,7.825,148.288
C05108=1221.011,385.756,-78.071,-175.793,7.827,148.288
C05109=1221.008,386.004,-78.104,-175.792,7.830,148.289
C05110=1221.004,386.251,-78.138,-175.791,7.833,148.289
C05111=1220.999,386.499,-78.173,-175.790,7.836,148.290
C05112=1220.995,386.746,-78.206,-175.790,7.838,148.290
C05113=1220.992,386.994,-78.240,-175.789,7.840,148.290
C05114=1220.987,387.242,-78.274,-175.787,7.843,148.291
C05115=1220.983,387.489,-78.308,-175.787,7.845,148.291
C05116=1220.978,387.737,-78.342,-175.786,7.848,148.292
C05117=1220.975,387.985,-78.376,-175.785,7.851,148.292
C05118=1220.971,388.232,-78.410,-175.784,7.853,148.292
C05119=1220.967,388.480,-78.444,-175.783,7.856,148.293
C05120=1220.962,388.727,-78.477,-175.782,7.859,148.293
C05121=1220.958,388.976,-78.512,-175.782,7.861,148.294
C05122=1220.954,389.223,-78.545,-175.780,7.864,148.294
C05123=1220.950,389.471,-78.580,-175.780,7.866,148.295
C05124=1220.946,389.719,-78.614,-175.779,7.869,148.295
C05125=1220.943,389.966,-78.648,-175.778,7.872,148.295
C05126=1220.938,390.214,-78.682,-175.777,7.874,148.296
C05127=1220.934,390.461,-78.715,-175.776,7.877,148.296
C05128=1220.930,390.709,-78.750,-175.775,7.880,148.297
C05129=1220.926,390.957,-78.783,-175.775,7.882,148.297
C05130=1220.921,391.204,-78.818,-175.774,7.885,148.298
C05131=1220.918,391.452,-78.852,-175.773,7.887,148.298
C05132=1220.913,391.699,-78.887,-175.772,7.890,148.298
C05133=1220.909,391.947,-78.920,-175.772,7.892,148.299
C05134=1220.905,392.195,-78.955,-175.771,7.895,148.299
C05135=1220.902,392.442,-78.988,-175.770,7.898,148.300
C05136=1220.897,392.724,-79.027,-175.769,7.900,148.300
C05137=1220.892,393.006,-79.066,-175.768,7.903,148.301
C05138=1220.888,393.288,-79.104,-175.767,7.906,148.301
C05139=1220.883,393.569,-79.144,-175.766,7.909,148.302
C05140=1220.879,393.817,-79.177,-175.766,7.912,148.302
C05141=1220.875,394.065,-79.212,-175.765,7.914,148.303
C05142=1220.871,394.312,-79.245,-175.764,7.916,148.303
C05143=1220.866,394.560,-79.280,-175.764,7.919,148.304
C05144=1220.863,394.808,-79.314,-175.762,7.922,148.304
C05145=1220.859,395.055,-79.349,-175.762,7.924,148.304
C05146=1220.854,395.302,-79.383,-175.761,7.927,148.305
C05147=1220.851,395.550,-79.417,-175.760,7.929,148.305
C05148=1220.846,395.798,-79.451,-175.760,7.932,148.306
C05149=1220.842,396.045,-79.485,-175.759,7.934,148.306
C05150=1220.838,396.294,-79.520,-175.758,7.936,148.307
C05151=1220.834,396.541,-79.554,-175.758,7.939,148.307
C05152=1220.830,396.788,-79.588,-175.757,7.941,148.308
C05153=1220.826,397.036,-79.622,-175.756,7.944,148.308
C05154=1220.822,397.283,-79.657,-175.756,7.946,148.308
C05155=1220.818,397.532,-79.691,-175.754,7.949,148.309
C05156=1220.814,397.779,-79.725,-175.754,7.951,148.309
C05157=1220.809,398.027,-79.759,-175.753,7.954,148.310
C05158=1220.806,398.274,-79.794,-175.752,7.956,148.310
C05159=1220.801,398.522,-79.828,-175.752,7.958,148.311
C05160=1220.797,398.769,-79.862,-175.751,7.961,148.311
C05161=1220.794,399.017,-79.897,-175.751,7.963,148.312
C05162=1220.789,399.264,-79.931,-175.750,7.965,148.312
C05163=1220.786,399.512,-79.965,-175.749,7.968,148.312
C05164=1220.781,399.760,-80.000,-175.749,7.970,148.313
C05165=1220.777,400.007,-80.034,-175.748,7.973,148.313
C05166=1220.773,400.255,-80.069,-175.747,7.975,148.314
C05167=1220.769,400.502,-80.103,-175.747,7.977,148.314
C05168=1220.765,400.749,-80.137,-175.746,7.980,148.315
C05169=1220.761,400.998,-80.172,-175.745,7.982,148.315
C05170=1220.756,401.245,-80.206,-175.745,7.984,148.315
C05171=1220.753,401.493,-80.240,-175.744,7.987,148.316
C05172=1220.749,401.740,-80.275,-175.743,7.989,148.316
C05173=1220.744,401.988,-80.309,-175.743,7.992,148.317
C05174=1220.741,402.235,-80.344,-175.742,7.994,148.317
C05175=1220.736,402.483,-80.378,-175.741,7.996,148.318
C05176=1220.732,402.731,-80.413,-175.741,7.999,148.318
C05177=1220.729,402.978,-80.447,-175.740,8.002,148.319
C05178=1220.725,403.226,-80.482,-175.740,8.004,148.319
C05179=1220.720,403.474,-80.516,-175.739,8.006,148.319
C05180=1220.716,403.721,-80.550,-175.738,8.009,148.320
C05181=1220.712,403.969,-80.585,-175.738,8.011,148.320
C05182=1220.708,404.216,-80.619,-175.738,8.013,148.321
C05183=1220.704,404.464,-80.653,-175.737,8.015,148.321
C05184=1220.700,404.711,-80.688,-175.736,8.018,148.322
C05185=1220.696,404.960,-80.723,-175.736,8.020,148.322
C05186=1220.692,405.207,-80.757,-175.735,8.022,148.323
C05187=1220.688,405.454,-80.792,-175.735,8.024,148.323
C05188=1220.684,405.702,-80.827,-175.734,8.027,148.324
C05189=1220.680,405.949,-80.861,-175.733,8.030,148.324
C05190=1220.676,406.197,-80.895,-175.733,8.032,148.324
C05191=1220.671,406.444,-80.930,-175.732,8.033,148.325
C05192=1220.667,406.692,-80.965,-175.731,8.037,148.325
C05193=1220.664,406.940,-80.999,-175.731,8.039,148.326
C05194=1220.660,407.188,-81.033,-175.731,8.041,148.326
C05195=1220.655,407.434,-81.069,-175.730,8.043,148.327
C05196=1220.651,407.683,-81.103,-175.730,8.045,148.327
C05197=1220.648,407.930,-81.137,-175.728,8.048,148.327
C05198=1220.643,408.177,-81.172,-175.728,8.050,148.328
C05199=1220.639,408.425,-81.207,-175.728,8.052,148.328
C05200=1220.634,408.673,-81.241,-175.727,8.054,148.329
C05201=1220.632,408.920,-81.276,-175.727,8.056,148.329
C05202=1220.627,409.167,-81.310,-175.726,8.059,148.330
C05203=1220.623,409.415,-81.345,-175.725,8.061,148.330
C05204=1220.618,409.663,-81.380,-175.725,8.063,148.331
C05205=1220.615,409.911,-81.414,-175.725,8.066,148.331
C05206=1220.611,410.157,-81.449,-175.724,8.068,148.331
C05207=1220.607,410.406,-81.484,-175.724,8.070,148.332
C05208=1220.602,410.653,-81.518,-175.723,8.073,148.332
C05209=1220.599,410.901,-81.553,-175.722,8.075,148.333
C05210=1220.595,411.148,-81.588,-175.722,8.077,148.333
C05211=1220.591,411.396,-81.623,-175.721,8.079,148.334
C05212=1220.586,411.643,-81.657,-175.721,8.081,148.334
C05213=1220.582,411.891,-81.692,-175.720,8.083,148.334
C05214=1220.579,412.138,-81.727,-175.720,8.086,148.335
C05215=1220.575,412.386,-81.761,-175.719,8.088,148.335
C05216=1220.570,412.633,-81.796,-175.718,8.090,148.336
C05217=1220.566,412.881,-81.831,-175.718,8.093,148.336
C05218=1220.562,413.128,-81.866,-175.717,8.095,148.337
C05219=1220.559,413.376,-81.900,-175.717,8.097,148.337
C05220=1220.554,413.623,-81.935,-175.717,8.099,148.337
C05221=1220.550,413.871,-81.969,-175.716,8.101,148.338
C05222=1220.546,414.118,-82.005,-175.716,8.103,148.338
C05223=1220.542,414.366,-82.039,-175.715,8.105,148.339
C05224=1220.538,414.614,-82.074,-175.715,8.107,148.339
C05225=1220.535,414.861,-82.109,-175.714,8.109,148.340
C05226=1220.530,415.108,-82.143,-175.714,8.112,148.340
C05227=1220.526,415.357,-82.178,-175.713,8.114,148.340
C05228=1220.523,415.573,-82.209,-175.713,8.115,148.341
C05229=1220.520,415.790,-82.239,-175.713,8.118,148.341
C05230=1220.515,416.007,-82.270,-175.712,8.120,148.342
C05231=1220.512,416.223,-82.300,-175.711,8.122,148.342
C05232=1220.509,416.440,-82.331,-175.711,8.124,148.342
C05233=1220.505,416.657,-82.362,-175.711,8.125,148.343
C05234=1220.502,416.874,-82.392,-175.710,8.127,148.343
C05235=1220.502,417.090,-82.422,-175.710,8.129,148.343
C05236=1220.080,417.091,-82.457,-175.713,8.139,148.347
C05237=1220.080,416.873,-82.426,-175.713,8.137,148.347
C05238=1220.083,416.654,-82.396,-175.714,8.135,148.346
C05239=1220.087,416.436,-82.365,-175.714,8.134,148.346
C05240=1220.090,416.218,-82.334,-175.715,8.132,148.346
C05241=1220.094,416.000,-82.303,-175.715,8.130,148.345
C05242=1220.097,415.782,-82.273,-175.716,8.128,148.345
C05243=1220.101,415.564,-82.242,-175.716,8.126,148.345
C05244=1220.105,415.346,-82.212,-175.717,8.124,148.344
C05245=1220.109,415.098,-82.177,-175.717,8.122,148.344
C05246=1220.113,414.851,-82.142,-175.718,8.120,148.343
C05247=1220.116,414.603,-82.107,-175.718,8.118,148.343
C05248=1220.121,414.356,-82.073,-175.718,8.116,148.342
C05249=1220.124,414.108,-82.037,-175.719,8.113,148.342
C05250=1220.129,413.861,-82.003,-175.719,8.111,148.342
C05251=1220.133,413.613,-81.968,-175.720,8.109,148.341
C05252=1220.137,413.366,-81.933,-175.720,8.107,148.341
C05253=1220.140,413.118,-81.899,-175.721,8.105,148.340
C05254=1220.144,412.870,-81.864,-175.721,8.103,148.340
C05255=1220.149,412.623,-81.829,-175.722,8.101,148.339
C05256=1220.153,412.375,-81.794,-175.722,8.098,148.339
C05257=1220.157,412.127,-81.759,-175.723,8.096,148.339
C05258=1220.160,411.880,-81.725,-175.724,8.094,148.338
C05259=1220.165,411.633,-81.690,-175.724,8.092,148.338
C05260=1220.169,411.385,-81.655,-175.725,8.090,148.337
C05261=1220.173,411.137,-81.621,-175.725,8.087,148.337
C05262=1220.177,410.889,-81.586,-175.725,8.085,148.336
C05263=1220.181,410.643,-81.551,-175.726,8.083,148.336
C05264=1220.185,410.395,-81.516,-175.727,8.080,148.336
C05265=1220.189,410.147,-81.482,-175.727,8.078,148.335
C05266=1220.193,409.899,-81.447,-175.728,8.076,148.335
C05267=1220.197,409.653,-81.412,-175.728,8.074,148.334
C05268=1220.201,409.405,-81.378,-175.728,8.072,148.334
C05269=1220.205,409.157,-81.343,-175.729,8.070,148.333
C05270=1220.210,408.910,-81.309,-175.730,8.067,148.333
C05271=1220.214,408.661,-81.274,-175.730,8.065,148.332
C05272=1220.217,408.415,-81.239,-175.731,8.062,148.332
C05273=1220.221,408.167,-81.204,-175.731,8.061,148.332
C05274=1220.226,407.919,-81.170,-175.731,8.058,148.331
C05275=1220.229,407.672,-81.136,-175.733,8.055,148.331
C05276=1220.234,407.424,-81.101,-175.733,8.053,148.330
C05277=1220.238,407.176,-81.066,-175.734,8.051,148.330
C05278=1220.242,406.929,-81.031,-175.734,8.049,148.329
C05279=1220.245,406.681,-80.997,-175.734,8.047,148.329
C05280=1220.250,406.434,-80.962,-175.736,8.044,148.329
C05281=1220.254,406.186,-80.928,-175.736,8.042,148.328
C05282=1220.258,405.939,-80.893,-175.736,8.040,148.328
C05283=1220.262,405.691,-80.859,-175.737,8.038,148.327
C05284=1220.266,405.443,-80.824,-175.738,8.035,148.327
C05285=1220.271,405.196,-80.790,-175.738,8.033,148.326
C05286=1220.273,404.949,-80.755,-175.739,8.031,148.326
C05287=1220.278,404.701,-80.721,-175.739,8.029,148.325
C05288=1220.282,404.453,-80.686,-175.740,8.025,148.325
C05289=1220.286,404.206,-80.652,-175.741,8.023,148.325
C05290=1220.290,403.958,-80.617,-175.741,8.021,148.324
C05291=1220.294,403.711,-80.583,-175.741,8.019,148.324
C05292=1220.299,403.463,-80.548,-175.742,8.016,148.323
C05293=1220.302,403.215,-80.514,-175.743,8.014,148.323
C05294=1220.307,402.968,-80.479,-175.743,8.012,148.322
C05295=1220.311,402.720,-80.445,-175.744,8.009,148.322
C05296=1220.315,402.473,-80.411,-175.745,8.007,148.321
C05297=1220.318,402.225,-80.376,-175.745,8.005,148.321
C05298=1220.323,401.977,-80.341,-175.746,8.002,148.321
C05299=1220.327,401.730,-80.308,-175.746,8.000,148.320
C05300=1220.331,401.482,-80.273,-175.747,7.998,148.320
C05301=1220.335,401.235,-80.239,-175.748,7.995,148.319
C05302=1220.339,400.987,-80.204,-175.748,7.993,148.319
C05303=1220.343,400.739,-80.170,-175.749,7.991,148.318
C05304=1220.347,400.492,-80.136,-175.750,7.988,148.318
C05305=1220.351,400.244,-80.101,-175.750,7.986,148.317
C05306=1220.356,399.997,-80.066,-175.751,7.983,148.317
C05307=1220.359,399.749,-80.032,-175.752,7.981,148.316
C05308=1220.363,399.501,-79.998,-175.752,7.978,148.316
C05309=1220.368,399.254,-79.963,-175.753,7.976,148.316
C05310=1220.371,399.006,-79.929,-175.754,7.973,148.315
C05311=1220.376,398.759,-79.895,-175.754,7.971,148.315
C05312=1220.380,398.512,-79.861,-175.755,7.968,148.314
C05313=1220.384,398.263,-79.826,-175.755,7.966,148.314
C05314=1220.388,398.016,-79.791,-175.756,7.964,148.313
C05315=1220.391,397.768,-79.757,-175.757,7.961,148.313
C05316=1220.396,397.521,-79.723,-175.757,7.959,148.312
C05317=1220.400,397.274,-79.689,-175.759,7.956,148.312
C05318=1220.404,397.026,-79.654,-175.759,7.954,148.311
C05319=1220.408,396.778,-79.621,-175.760,7.951,148.311
C05320=1220.412,396.530,-79.586,-175.761,7.949,148.311
C05321=1220.416,396.282,-79.551,-175.761,7.947,148.310
C05322=1220.420,396.035,-79.518,-175.762,7.944,148.310
C05323=1220.425,395.788,-79.483,-175.762,7.942,148.309
C05324=1220.428,395.540,-79.449,-175.763,7.939,148.309
C05325=1220.433,395.293,-79.414,-175.764,7.937,148.309
C05326=1220.436,395.045,-79.380,-175.765,7.934,148.308
C05327=1220.441,394.797,-79.346,-175.765,7.932,148.308
C05328=1220.445,394.550,-79.313,-175.767,7.929,148.307
C05329=1220.449,394.301,-79.278,-175.767,7.927,148.307
C05330=1220.452,394.054,-79.244,-175.768,7.924,148.306
C05331=1220.457,393.807,-79.209,-175.768,7.922,148.306
C05332=1220.460,393.559,-79.176,-175.769,7.919,148.305
C05333=1220.465,393.277,-79.136,-175.771,7.916,148.305
C05334=1220.469,392.996,-79.098,-175.771,7.913,148.304
C05335=1220.475,392.713,-79.059,-175.771,7.911,148.304
C05336=1220.479,392.432,-79.020,-175.773,7.908,148.303
C05337=1220.484,392.184,-78.986,-175.774,7.905,148.303
C05338=1220.488,391.937,-78.952,-175.775,7.902,148.302
C05339=1220.491,391.689,-78.918,-175.775,7.900,148.302
C05340=1220.495,391.442,-78.884,-175.776,7.897,148.302
C05341=1220.500,391.194,-78.850,-175.777,7.895,148.301
C05342=1220.503,390.946,-78.816,-175.778,7.892,148.301
C05343=1220.508,390.698,-78.781,-175.778,7.890,148.300
C05344=1220.512,390.451,-78.747,-175.779,7.887,148.300
C05345=1220.516,390.202,-78.713,-175.780,7.884,148.299
C05346=1220.520,389.955,-78.679,-175.781,7.882,148.299
C05347=1220.525,389.708,-78.645,-175.782,7.879,148.298
C05348=1220.529,389.460,-78.612,-175.782,7.877,148.298
C05349=1220.532,389.212,-78.577,-175.783,7.874,148.298
C05350=1220.536,388.965,-78.543,-175.785,7.871,148.297
C05351=1220.541,388.717,-78.510,-175.785,7.869,148.297
C05352=1220.545,388.469,-78.475,-175.786,7.866,148.296
C05353=1220.548,388.222,-78.441,-175.787,7.864,148.296
C05354=1220.553,387.974,-78.407,-175.787,7.861,148.295
C05355=1220.557,387.727,-78.374,-175.789,7.858,148.295
C05356=1220.560,387.479,-78.339,-175.790,7.856,148.295
C05357=1220.565,387.231,-78.306,-175.790,7.854,148.294
C05358=1220.569,386.984,-78.272,-175.792,7.851,148.294
C05359=1220.574,386.736,-78.238,-175.792,7.848,148.293
C05360=1220.577,386.488,-78.204,-175.793,7.846,148.293
C05361=1220.581,386.241,-78.170,-175.794,7.843,148.293
C05362=1220.586,385.993,-78.136,-175.795,7.840,148.292
C05363=1220.590,385.746,-78.102,-175.796,7.837,148.292
C05364=1220.593,385.497,-78.069,-175.797,7.835,148.291
C05365=1220.598,385.250,-78.034,-175.798,7.832,148.291
C05366=1220.602,385.002,-78.001,-175.799,7.829,148.290
C05367=1220.606,384.755,-77.967,-175.800,7.827,148.290
C05368=1220.610,384.507,-77.932,-175.800,7.824,148.289
C05369=1220.614,384.259,-77.899,-175.802,7.821,148.289
C05370=1220.618,384.012,-77.865,-175.803,7.819,148.289
C05371=1220.623,383.764,-77.832,-175.803,7.817,148.288
C05372=1220.626,383.517,-77.798,-175.805,7.814,148.288
C05373=1220.630,383.269,-77.764,-175.806,7.811,148.288
C05374=1220.635,383.021,-77.730,-175.806,7.808,148.287
C05375=1220.639,382.773,-77.697,-175.808,7.805,148.287
C05376=1220.642,382.526,-77.663,-175.808,7.803,148.286
C05377=1220.647,382.278,-77.629,-175.810,7.800,148.286
C05378=1220.651,382.030,-77.595,-175.811,7.797,148.285
C05379=1220.655,381.783,-77.562,-175.812,7.795,148.285
C05380=1220.660,381.535,-77.528,-175.813,7.792,148.285
C05381=1220.663,381.288,-77.494,-175.814,7.790,148.284
C05382=1220.667,381.039,-77.460,-175.814,7.787,148.284
C05383=1220.671,380.792,-77.427,-175.816,7.784,148.283
C05384=1220.676,380.544,-77.393,-175.817,7.781,148.283
C05385=1220.680,380.296,-77.360,-175.818,7.778,148.282
C05386=1220.684,380.049,-77.326,-175.819,7.775,148.282
C05387=1220.688,379.801,-77.293,-175.820,7.773,148.282
C05388=1220.692,379.553,-77.258,-175.821,7.771,148.281
C05389=1220.696,379.306,-77.225,-175.822,7.768,148.281
C05390=1220.700,379.058,-77.191,-175.823,7.765,148.281
C05391=1220.704,378.811,-77.158,-175.825,7.762,148.280
C05392=1220.709,378.563,-77.124,-175.826,7.759,148.280
C05393=1220.713,378.315,-77.091,-175.827,7.757,148.279
C05394=1220.716,378.067,-77.056,-175.828,7.754,148.279
C05395=1220.720,377.819,-77.023,-175.829,7.751,148.279
C05396=1220.724,377.572,-76.990,-175.830,7.748,148.278
C05397=1220.729,377.324,-76.956,-175.831,7.746,148.278
C05398=1220.733,377.077,-76.922,-175.832,7.743,148.277
C05399=1220.737,376.829,-76.889,-175.833,7.741,148.277
C05400=1220.741,376.581,-76.856,-175.835,7.738,148.277
C05401=1220.745,376.333,-76.822,-175.836,7.735,148.276
C05402=1220.749,376.086,-76.789,-175.837,7.732,148.276
C05403=1220.754,375.838,-76.755,-175.838,7.729,148.275
C05404=1220.758,375.590,-76.722,-175.839,7.726,148.275
C05405=1220.762,375.343,-76.688,-175.840,7.724,148.275
C05406=1220.766,375.095,-76.655,-175.842,7.721,148.274
C05407=1220.770,374.847,-76.622,-175.843,7.718,148.274
C05408=1220.774,374.600,-76.589,-175.844,7.715,148.274
C05409=1220.778,374.351,-76.555,-175.846,7.713,148.273
C05410=1220.782,374.104,-76.521,-175.847,7.710,148.273
C05411=1220.786,373.856,-76.487,-175.848,7.707,148.273
C05412=1220.790,373.608,-76.454,-175.849,7.704,148.272
C05413=1220.795,373.360,-76.421,-175.850,7.701,148.272
C05414=1220.799,373.113,-76.388,-175.852,7.699,148.271
C05415=1220.803,372.865,-76.355,-175.853,7.696,148.271
C05416=1220.807,372.617,-76.322,-175.854,7.693,148.271
C05417=1220.811,372.370,-76.288,-175.856,7.690,148.270
C05418=1220.815,372.122,-76.255,-175.857,7.688,148.270
C05419=1220.819,371.875,-76.221,-175.858,7.685,148.270
C05420=1220.824,371.627,-76.188,-175.859,7.682,148.269
C05421=1220.827,371.378,-76.154,-175.861,7.679,148.269
C05422=1220.832,371.131,-76.121,-175.862,7.677,148.269
C05423=1220.836,370.883,-76.088,-175.863,7.674,148.268
C05424=1220.840,370.635,-76.055,-175.864,7.671,148.268
C05425=1220.844,370.387,-76.022,-175.866,7.668,148.268
C05426=1220.848,370.140,-75.988,-175.868,7.665,148.267
C05427=1220.852,369.892,-75.955,-175.869,7.662,148.267
C05428=1220.856,369.644,-75.922,-175.870,7.659,148.266
C05429=1220.861,369.396,-75.889,-175.872,7.657,148.266
C05430=1220.865,369.149,-75.856,-175.873,7.654,148.266
C05431=1220.869,368.901,-75.823,-175.874,7.651,148.265
C05432=1220.873,368.653,-75.789,-175.876,7.648,148.265
C05433=1220.877,368.405,-75.756,-175.877,7.646,148.265
C05434=1220.881,368.158,-75.723,-175.878,7.643,148.264
C05435=1220.885,367.910,-75.690,-175.880,7.640,148.264
C05436=1220.890,367.662,-75.657,-175.881,7.637,148.264
C05437=1220.894,367.383,-75.619,-175.883,7.634,148.263
C05438=1220.899,367.103,-75.582,-175.885,7.630,148.263
C05439=1220.904,366.823,-75.545,-175.886,7.628,148.263
C05440=1220.908,366.543,-75.507,-175.888,7.624,148.262
C05441=1220.912,366.295,-75.474,-175.889,7.621,148.262
C05442=1220.916,366.047,-75.441,-175.890,7.619,148.262
C05443=1220.920,365.799,-75.408,-175.892,7.616,148.261
C05444=1220.924,365.551,-75.376,-175.893,7.613,148.261
C05445=1220.928,365.304,-75.343,-175.895,7.610,148.261
C05446=1220.933,365.057,-75.310,-175.897,7.607,148.261
C05447=1220.937,364.809,-75.277,-175.898,7.604,148.260
C05448=1220.941,364.561,-75.243,-175.899,7.602,148.260
C05449=1220.945,364.313,-75.210,-175.901,7.599,148.260
C05450=1220.949,364.065,-75.178,-175.902,7.596,148.259
C05451=1220.954,363.817,-75.145,-175.904,7.593,148.259
C05452=1220.958,363.570,-75.112,-175.906,7.590,148.259
C05453=1220.961,363.322,-75.079,-175.907,7.587,148.258
C05454=1220.966,363.074,-75.047,-175.908,7.585,148.258
C05455=1220.970,362.826,-75.013,-175.910,7.581,148.258
C05456=1220.974,362.578,-74.980,-175.912,7.579,148.258
C05457=1220.978,362.331,-74.947,-175.913,7.576,148.257
C05458=1220.982,362.082,-74.915,-175.915,7.573,148.257
C05459=1220.986,361.835,-74.882,-175.916,7.571,148.257
C05460=1220.990,361.587,-74.849,-175.918,7.567,148.256
C05461=1220.994,361.339,-74.816,-175.919,7.564,148.256
C05462=1220.999,361.091,-74.783,-175.921,7.562,148.256
C05463=1221.003,360.843,-74.750,-175.922,7.559,148.256
C05464=1221.006,360.596,-74.718,-175.924,7.556,148.255
C05465=1221.011,360.348,-74.686,-175.926,7.553,148.255
C05466=1221.015,360.101,-74.652,-175.927,7.550,148.255
C05467=1221.019,359.853,-74.619,-175.929,7.548,148.254
C05468=1221.024,359.605,-74.587,-175.931,7.544,148.254
